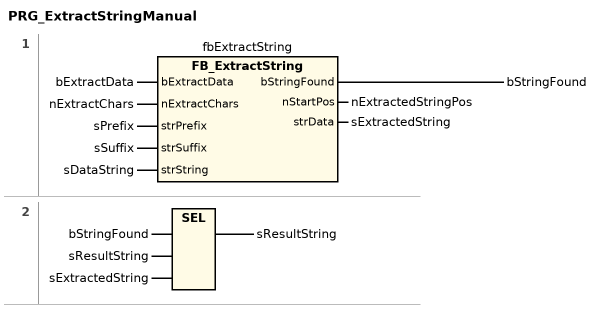
// NETWORK 1
fbExtractString(
    bExtractData := bExtractData,
    nExtractChars := nExtractChars,
    strPrefix := sPrefix,
    strSuffix := sSuffix,
    strString := sDataString,
    nStartPos => nExtractedStringPos,
    strData => sExtractedString); // FB_ExtractString
bStringFound := fbExtractString.bStringFound;

// NETWORK 2
sResultString := SEL(bStringFound, sResultString, sExtractedString);

END_PROGRAM

// ---- POUs/TcUnit/FUN_ReplaceLongSingleCharTests/PRG_ReplaceLongSingleCharManual.TcPOU
PROGRAM PRG_ReplaceLongSingleCharManual
VAR
	
	sFullCode		: T_LongSTRING := 'ST=53;$02CT=10;DS=GZDNP5JOA3IL$1D;OG=3;XP=-50;YP=50;AP=-88;CS=06.2;SC=0070;QS=3;PN=1;$03$04
											ST=53;$02CT=10;DS=N7E1Y89UNK3O$1D;OG=3;XP=-50;YP=-50;AP=-88;CS=06.2;SC=0070;QS=3;PN=2;$03$04
											ST=53;$02CT=10;DS=JHWJXYFNX9DS$1D;OG=3;XP=50;YP=50;AP=-88;CS=06.2;SC=0070;QS=3;PN=3;$03$04
											ST=53;$02CT=10;DS=XGBEZLBV8A9I$1D;OG=3;XP=50;YP=-50;AP=-88;CS=06.2;SC=0070;QS=3;PN=4;$03$04'; 
	sCharRemove		: T_Char := '$1D';
	sReplacmentChar	: T_Char := '';
	
	sResult			: T_LongSTRING;
END_VAR

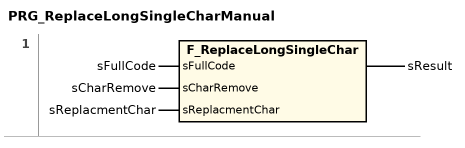
// NETWORK 1
sResult := F_ReplaceLongSingleChar(sFullCode := sFullCode, sCharRemove := sCharRemove, sReplacmentChar := sReplacmentChar);

END_PROGRAM

// ---- POUs/TcUnit/FB_LOGHandlerTests/PRG_LogHandlerManual.TcPOU
PROGRAM PRG_LogHandlerManual
VAR
	fbLogHandler			: FB_LOG_Handler;

	bLogData				: BOOL;
	sLogMessage				: T_LongSTRING;
	
	stEventDataUT				: ST_LOG_EventData;
	
	sResultMessage				: T_LongSTRING;
	
	bDone					: BOOL;
	bBufferOverflow			: BOOL;
END_VAR

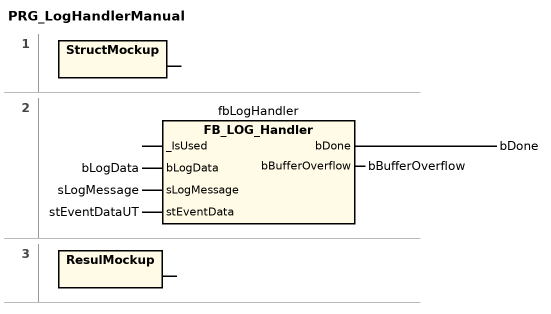
// NETWORK 1
StructMockup();

// NETWORK 2
fbLogHandler(
    bLogData := bLogData,
    sLogMessage := sLogMessage,
    stEventData := stEventDataUT,
    bBufferOverflow => bBufferOverflow); // FB_LOG_Handler
bDone := fbLogHandler.bDone;

// NETWORK 3
ResulMockup();

ACTION ResulMockup:
IF stEventDataUT.nImageByte < SIZEOF(sResultMessage) THEN
	MEMMOVE(ADR(sResultMessage), ADR(stEventDataUT.aDataLogImage), stEventDataUT.nImageByte);
END_IF
END_ACTION

ACTION StructMockup:

stEventDataUT.bEnable := gDevice.stMetsStatus.bSystemTimeValid;
stEventDataUT.sTimeStamp :=MID( F_SYSTEM_SystemTimeAsISO8601(gDevice.stMetsStatus.stCTDateTime.sSystemTime, gDevice.stMetsStatus.stCTDateTime.sUTCTimeZoneOffset ), 12, 12);

sLogMessage := '$01ST=53;$02CT=10;DS=GZDNP5JOA3IL;OG=3;XP=-50;YP=50;AP=-88;CS=06.2;SC=0070;QS=3;PN=1;$03
					$01ST=53;$02CT=10;DS=N7E1Y89UNK3O;OG=3;XP=-50;YP=-50;AP=-88;CS=06.2;SC=0070;QS=3;PN=2;$03
					$01ST=53;$02CT=10;DS=JHWJXYFNX9DS;OG=3;XP=50;YP=50;AP=-88;CS=06.2;SC=0070;QS=3;PN=3;$03
					$01ST=53;$02CT=10;DS=XGBEZLBV8A9I;OG=3;XP=50;YP=-50;AP=-88;CS=06.2;SC=0070;QS=3;PN=4;$03';
END_ACTION

END_PROGRAM

// ---- POUs/METS/Common LIB/08_SOFTWARE LIB/AI Codes And Validation FBs/F_CODE_GetItemAI.TcPOU
FUNCTION F_CODE_GetItemAI : T_MaxString
VAR_INPUT
	sFullCode		: T_MaxString;
	eCodeType		: E_CodeAI;
	stCodeInfo		: ST_CodeInfo;
END_VAR
VAR
	stItem			: ST_CodeValidation;
	
	sTemp			: T_MaxString;
	nStart			: INT;
	nEnd			: INT;
	
	sResultString	: T_MaxString;
END_VAR

IF stCodeInfo.nEntireLength > 0 THEN

	IF eCodeType = E_CodeAI.GTIN THEN 			stItem := stCodeInfo.stGTIN;
	ELSIF eCodeType = E_CodeAI.BATCH THEN 		stItem := stCodeInfo.stBatchID;
	ELSIF eCodeType = E_CodeAI.SERIAL THEN		stItem := stCodeInfo.stSerialCode;
	ELSIF eCodeType = E_CodeAI.PO THEN			stItem := stCodeInfo.stProductionOrder;
	ELSIF eCodeType = E_CodeAI.CRYPTO THEN		stItem := stCodeInfo.stCryptoCode;
	ELSIF eCodeType = E_CodeAI.RSKU THEN		stItem := stCodeInfo.stRSKU;
	ELSIF eCodeType = E_CodeAI.MRP THEN			stItem := stCodeInfo.stMRP;
	ELSIF eCodeType = E_CodeAI.BRANDSPEC THEN	stItem := stCodeInfo.stBrandSpecification;
	ELSIF eCodeType = E_CodeAI.PRODDATE THEN	stItem := stCodeInfo.stProduceDate;
	ELSIF eCodeType = E_CodeAI.USERFIELD THEN	stItem := stCodeInfo.stUserField3;
	END_IF

/////////////////////////////////////////////////////////////////////////////////////////////////////

	IF stItem.sStartAI <> '' AND stItem.sEndAI <> '' THEN
		
		nStart := FIND(sFullCode, stItem.sStartAI) + LEN(stItem.sStartAI);
		
		IF nStart > 0 THEN
			sTemp := RIGHT(sFullCode, LEN(sFullCode) - (nStart - 1));
		ELSE
			sTemp := sFullCode;
		END_IF
		
		nEnd := FIND(sTemp, stItem.sEndAI);
		
		IF nEnd = 0 THEN
			nEnd := LEN(sFullCode)+1;
		ELSE
			nEnd := nEnd +(nStart - 1);
		END_IF
		
	ELSIF stItem.sStartAI <> '' AND stItem.nCodeLength > 0 THEN
		
		nStart := FIND(sFullCode, stItem.sStartAI) + LEN(stItem.sStartAI);
		nEnd := nStart + stItem.nCodeLength;
		
	ELSIF stItem.nCodeStartPos > 0 AND stItem.sEndAI <> '' THEN
		
		nStart := stItem.nCodeStartPos;
		sTemp := RIGHT(sFullCode, LEN(sFullCode) - (nStart - 1));
		nEnd := FIND(sTemp, stItem.sEndAI);
		
		IF nEnd = 0 THEN
			nEnd := LEN(sFullCode)+1;
		ELSE
			nEnd := nEnd +(nStart - 1);
		END_IF
		
	ELSIF stItem.nCodeStartPos >= 0 AND stItem.nCodeLength > 0 THEN
		
		nStart := stItem.nCodeStartPos;
		nEnd := nStart + stItem.nCodeLength;
	ELSE
		nStart := 0;
		nEnd := 0;
	END_IF
	
	IF nStart > 0 AND nEnd > 0 THEN
		sResultString := MID(sFullCode, nEnd - nStart, nStart);
	ELSE
		sResultString := '';
	END_IF
ELSE
	sResultString := '';
END_IF

F_CODE_GetItemAI := sResultString;

END_FUNCTION

// ---- POUs/METS/Common LIB/09_SYSTEM LIB/FB_SYSTEM_CoreFolders.TcPOU
FUNCTION_BLOCK FB_SYSTEM_CoreFolders
VAR_INPUT
	bExecute				: BOOL;		(* set TRUE to generate system folders *)
	sBasePath			: T_FolderName;	(* CaseTrace base folder path *)
	aBaseFolder			: ARRAY[1..cSYSTEM_FOLDER_LIMIT] OF T_FolderName;
END_VAR
VAR_OUTPUT
	bDone				: BOOL;		(* TRUE = system folders complete *)
	bBusy				: BOOL;		(* TRUE = system folders in progress *)
	bError				: BOOL;		(* TRUE = system folders error *)
	nErrorID				: UDINT;	(* error code *)
	bSystemFolderOK		: BOOL;		(* TRUE = system folders OK *)
	sStatus					: STRING(25);	(* system folder status *)

END_VAR
VAR
	fbExecute				: R_TRIG;
	eState				: E_SYSTEM_MaintainFolders;
	eErrorState			: E_SYSTEM_MaintainFolders;
	nMaxIndex			: INT;
	nIndex				: INT;
	eCmdType		: E_EnumCmdType;
	fbFindFolder		: FB_EnumFindFileEntry;
	fbCreateFolder			: FB_CreateDir;

END_VAR

(* rising edge of bExecute *)
fbExecute(CLK := bExecute);

CASE eState OF

	(* idle *)
	E_FOLDER_IDLE:

		(* rising edge of bExecute *)
		IF fbExecute.Q = TRUE THEN

			(* update outputs *)
			bDone := FALSE;
			bBusy := TRUE;
			bError := FALSE;
			nErrorID := 0;

			(* max number of BASE folders and start with 1st folder *)
			nMaxIndex := UDINT_TO_INT(SIZEOF(aBaseFolder) / SIZEOF(aBaseFolder[1]));
			nIndex := 1;
			eCmdType := eEnumCmd_First;

			//eState := E_FOLDER_CREATEBASEPATH;
			eState := E_FOLDER_ININT_CHECK;

		(* bExecute has been reset *)
		ELSIF bExecute = FALSE THEN

			(* reset outputs *)
			bDone := FALSE;
			bBusy := FALSE;
			bError := FALSE;
			nErrorID := 0;
		END_IF

	E_FOLDER_ININT_CHECK:
					eCmdType := eEnumCmd_First;
					eState := E_FOLDER_CHECK;
	
	E_FOLDER_CHECK:

		(* find folder *)
		fbFindFolder(
			sNetId		:= '',
			sPathName	:= CONCAT(sBasePath, aBaseFolder[nIndex]),
			eCmd		:= eCmdType,
			bExecute	:= TRUE,
			tTimeout	:= T#1s
		);

		(* find folder complete *)
		IF fbFindFolder.bBusy = FALSE THEN

			(* find folder completed OK *)
			IF fbFindFolder.bError = FALSE THEN

				(* folder found *)
				IF fbFindFolder.stFindFile.fileAttributes.bDirectory = TRUE THEN

				
						(* all BASE folders completed *)
				IF nIndex = nMaxIndex THEN

					eState := E_FOLDER_DONE;

				(* more BASE folders *)
				ELSE
					nIndex := nIndex + 1;
					eCmdType := eEnumCmd_Abort;
					eState := E_FOLDER_ININT_CHECK;
				END_IF

				(* end of list *)
				ELSIF fbFindFolder.bEOE = TRUE THEN

						eState := E_FOLDER_CREATEBASEPATH;
				END_IF

			(* find folder completed OK *)
			ELSE

				(* update outputs *)
				bError := TRUE;
				nErrorID := fbFindFolder.nErrID;
				eErrorState := eState;

				eState := E_FOLDER_DONE;
			END_IF

			(* close off fbFindFolder *)
			fbFindFolder(bExecute := FALSE);
		END_IF
		
	(* create BASE folders *)
	E_FOLDER_CREATEBASEPATH:

		(* create folder *)
		fbCreateFolder(
			sNetId		:= '',
			sPathName	:= CONCAT(sBasePath, aBaseFolder[nIndex]),
			ePath		:= PATH_GENERIC,
			bExecute	:= TRUE,
			tTimeout	:= T#1s
		);

		(* create folder complete *)
		IF fbCreateFolder.bBusy = FALSE THEN

			(* create folder completed OK or folder already exists *)
			IF fbCreateFolder.bError = FALSE OR (fbCreateFolder.bError = TRUE AND fbCreateFolder.nErrId = cFAILED_OBJECT_ALREADY_EXIST) THEN

				(* all BASE folders completed *)
				IF nIndex = nMaxIndex THEN

					eState := E_FOLDER_DONE;

				(* more BASE folders *)
				ELSE

					(* next BASE folder *)
					nIndex := nIndex + 1;
					eState := E_FOLDER_ININT_CHECK;
				END_IF

			(* create folder error *)
			ELSE

				(* no error active *)
				IF bError = FALSE THEN

					(* update outputs *)
					bError := TRUE;
					nErrorID := fbCreateFolder.nErrId;
					eErrorState := eState;
					sStatus := CONCAT(sBasePath, aBaseFolder[nIndex]);
				END_IF

				eState := E_FOLDER_DONE;
			END_IF

			(* close off fbCreateFolder *)
			fbCreateFolder(bExecute := FALSE);
		END_IF


	(* done *)
	E_FOLDER_DONE:

		(* no error occurred *)
		IF bError = FALSE THEN

			(* update status *)
			bSystemFolderOK 		:= TRUE;
			sStatus 				:= 'Core folders OK';
			
		ELSE
			(* update status *)
			bSystemFolderOK 		:= FALSE;
			sStatus 				:= 'Core folders NOT OK';
		END_IF

		(* update outputs *)
		bDone := TRUE;
		bBusy := FALSE;

		eState := E_FOLDER_IDLE;


(* unknown state *)
ELSE

	eState := E_FOLDER_IDLE;

	(* reset outputs *)
	bDone := FALSE;
	bBusy := FALSE;
	bError := FALSE;
	nErrorID := 0;
	bSystemFolderOK := FALSE;
	sStatus := '';
END_CASE

END_FUNCTION_BLOCK

// ---- POUs/METS/Common LIB/09_SYSTEM LIB/FB_SYSTEM_CorePaths.TcPOU
FUNCTION_BLOCK FB_SYSTEM_CorePaths
VAR_INPUT
	bExecute				: BOOL;		(* set TRUE to generate system folders *)
	sMETSAppPath				: T_FolderPath;
	sMETSLogsPath				: T_FolderPath;	
	sMETSProcessPath			: T_FolderPath;
	aCoreFolders			: ARRAY[1..cSYSTEM_FOLDER_LIMIT] OF T_FolderName;
	aAuxFolders				: ARRAY[1..cSYSTEM_FOLDER_LIMIT] OF T_FolderName;
END_VAR
VAR_OUTPUT
	sArchiveDBPath			: T_FolderPath;	(*local ArchiveDB path*)
	sBridgeAppPath 			: T_FolderPath;	(* local Bridge path *)
	sLoggerAppPath			: T_FolderPath;	(*  *)
	sWebHMIPath				: T_FolderPath;	(*  *)
	sDeleteArchivePath		: T_FolderPath;	(*  *)
	
	sPCMPath 			: T_FolderPath;	(* local PCM path *)
	sPCMIncomingPath 	: T_FolderPath;	(* local PCM/Incoming path *)
	sCHMPath 			: T_FolderPath;	(* local CHM path *)
	sSettingsPath		 	: T_FolderPath;	(* local Setting*)
	sBackupsPath			: T_FolderPath; (*local Setting/Backup path*)
	sRecipePath				: T_FolderPath; (*local Setting/Recipe path*)
	sCamerasPath				: T_FolderPath;	(* local Camera path *)
	sPrintersPath			: T_FolderPath;	(* local Camera path *)
	
	sOCVPath 			: T_FolderPath;	(* local OCV path *)
	sOACPath 			: T_FolderPath;	(* local OAC path *)
	sCACPath 			: T_FolderPath;	(* local CAC path *)
	sSystemLogPath			: T_FolderPath;	(* local Log path *)
	
END_VAR
VAR
	fbExecute				: R_TRIG;

END_VAR
(*
cMETS_CORE_FOLDERS					: ARRAY[1..cSYSTEM_FOLDER_LIMIT] OF T_FolderName :=[
			(*01*)'CHM\',		(*02*)'CHM\Archive\',		(*03*)'CHM\Error\',		(*04*)'CHM\OK\',		(*05*)'CHM\Commissioning_Mode\',	(*06*)'CHM\Restore\',
			(*07*)'PCM\',		(*08*)'PCM\Archive\',		(*09*)'PCM\Error\',		(*10*)'PCM\Incoming\',
			(*11*)'Settings\',	(*12*)'Settings\Backups\',	(*13*)'Settings\Recipe\',
			(*14*)'Cameras\',
			(*15*)'Printers\',	(*16*)'Printers\Templates'];
			
cMETS_AUX_FOLDERS					: ARRAY[1..cSYSTEM_FOLDER_LIMIT] OF T_FolderName :=[
			(*01*)'CAC\',		(*02*)'CAC\Archive\',		(*03*)'CAC\Error\',		(*04*)'CAC\Restored\',
			(*05*)'OAC\',		(*06*)'OAC\Error\',			(*07*)'OAC\Empty\',
			(*08*)'OCV\',		(*09*)'OCV\Error\',			(*10*)'OCV\Empty\',
			(*11*)'SystemLog\',
			(*12*)'ArchiveDB\',
			(*13*)'BridgeApp\Bridge_Core\',
			(*14*)'LoggerApp\Service\',
			(*15*)'WebHMI\',
			(*16*)'DeleteArchiveTool\'];
*)


(* rising edge of bExecute *)
fbExecute(CLK := bExecute);

(* rising edge of bExecute *)
IF fbExecute.Q = TRUE THEN

(* populate local folder paths *)
	sArchiveDBPath			:= CONCAT(sMETSAppPath, aAuxFolders[12]);
	sBridgeAppPath 			:= CONCAT(sMETSAppPath, aAuxFolders[13]);
	sLoggerAppPath			:= CONCAT(sMETSAppPath, aAuxFolders[14]);
	sWebHMIPath				:= CONCAT(sMETSAppPath, aAuxFolders[15]);
	sDeleteArchivePath		:= CONCAT(sMETSAppPath, aAuxFolders[16]);
	
	sPCMPath 				:= CONCAT(sMETSProcessPath, aCoreFolders[7]);
	sPCMIncomingPath 		:= CONCAT(sMETSProcessPath, aCoreFolders[10]);
	sCHMPath 				:= CONCAT(sMETSProcessPath, aCoreFolders[1]);
	sSettingsPath		 	:= CONCAT(sMETSProcessPath, aCoreFolders[11]);
	sBackupsPath			:= CONCAT(sMETSProcessPath, aCoreFolders[12]);
	sRecipePath				:= CONCAT(sMETSProcessPath, aCoreFolders[13]);
	sCamerasPath			:= CONCAT(sMETSProcessPath, aCoreFolders[14]);
	sPrintersPath			:= CONCAT(sMETSProcessPath, aCoreFolders[15]);
	
	sOCVPath 				:= CONCAT(sMETSProcessPath, aAuxFolders[8]);
	sOACPath 				:= CONCAT(sMETSProcessPath, aAuxFolders[5]);
	sCACPath 				:= CONCAT(sMETSProcessPath, aAuxFolders[1]);
	
	sSystemLogPath			:= CONCAT(sMETSLogsPath, aAuxFolders[11]);
			
ELSIF NOT bExecute THEN		
			
	(* populate local folder paths *)
	sArchiveDBPath			:='';
	sBridgeAppPath 			:='';
	sLoggerAppPath			:='';
	sWebHMIPath				:='';
	sDeleteArchivePath		:='';
	
	sPCMPath 				:='';
	sPCMIncomingPath 		:='';
	sCHMPath 				:='';
	sSettingsPath		 	:='';
	sBackupsPath			:='';
	sRecipePath				:='';
	sCamerasPath			:='';
	sPrintersPath			:='';
	
	sOCVPath 				:='';
	sOACPath 				:='';
	sCACPath 				:='';
	
	sSystemLogPath			:='';		
			
END_IF

END_FUNCTION_BLOCK

// ---- POUs/TcUnit/FB_CASE_ValidateContentTests/PRG_CASE_ValidateContentManual.TcPOU
PROGRAM PRG_CASE_ValidateContentManual
VAR
	fbCase_ValidateContent		: FB_CASE_ValidateContent;
	
	
	(* Init function/method declarations*)
	rTrigDataInit		: R_TRIG;
	bDataInit			: BOOL;
	iOuter				: INT;
	iPack				: INT;
	sPackNum			: STRING;
	sOuterNum			: STRING;
	sPackCode			: STRING;
	
	(* Inputs *)
	bExecute 					: BOOL;
	stCTDateTime				: ST_SYSTEM_DateTime;	(* CaseTrace date/time structure *)
	bIsDuplicateOuters			: BOOL;
	bIsDuplicatePacks			: BOOL;
	stOuterDataNotFound			: ST_RejectItems;
	stRejectReasonsForOuter		: ST_RejectReasonsForOuter;
	
	(* In/Out *)
	stProductInstruction		: ST_PCM_Status;
	nSecquentionalCounter		: UDINT;
	stCodeInfo_Outer			: ST_CodeInfo;
	stCaseRejectReasons			: ST_RejectReasonsForCase;
	stCACData 					: ST_CAC_Data;
	
	(* Outputs *)
	bDone 						: BOOL;
	bBusy						: BOOL;
	bError						: BOOL;
	nErrorID 					: UDINT;

	sRejectCode					: T_MaxString;
	nValidationIndex			: INT;
	
END_VAR

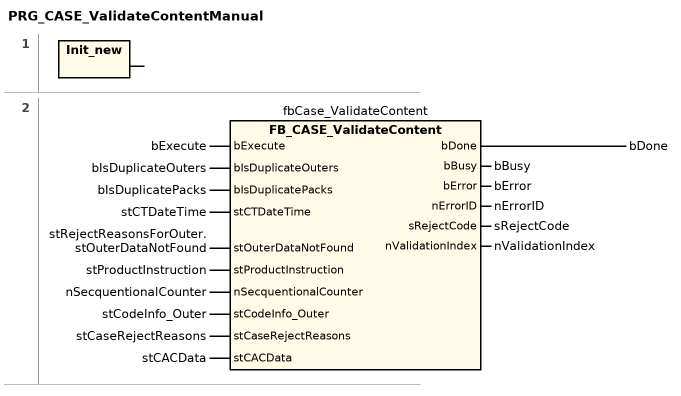
// NETWORK 1
Init_new();

// NETWORK 2
fbCase_ValidateContent(
    bExecute := bExecute,
    bIsDuplicateOuters := bIsDuplicateOuters,
    bIsDuplicatePacks := bIsDuplicatePacks,
    stCTDateTime := stCTDateTime,
    stOuterDataNotFound := stRejectReasonsForOuter.stOuterDataNotFound,
    stProductInstruction := stProductInstruction,
    nSecquentionalCounter := nSecquentionalCounter,
    stCodeInfo_Outer := stCodeInfo_Outer,
    stCaseRejectReasons := stCaseRejectReasons,
    stCACData := stCACData,
    bBusy => bBusy,
    bError => bError,
    nErrorID => nErrorID,
    sRejectCode => sRejectCode,
    nValidationIndex => nValidationIndex); // FB_CASE_ValidateContent
bDone := fbCase_ValidateContent.bDone;

ACTION Init:
rTrigDataInit(CLK := bDataInit);

IF rTrigDataInit.Q THEN
		
	stProductInstruction.nOutersPerCase		:= 50;
	stProductInstruction.nPacksPerOuter 	:= 10;











	FOR iOuter := 1 TO stProductInstruction.nOutersPerCase DO
		(* Ustaw outer *)
		stCACData.Outer[iOuter].Barcode    := CONCAT('OUTER', INT_TO_STRING(iOuter));
		stCACData.Outer[iOuter].OuterCodeStatus := 5;
		






		FOR iPack := 1 TO stProductInstruction.nPacksPerOuter DO
			(* Pack number z zerami *)
			sPackNum := CONCAT('0', INT_TO_STRING(iPack));  (* dla 1-9: '01'-'09' *)
			IF iPack = 10 THEN
				sPackNum := '10';
			END_IF;
			
			(* Outer number z zerami dla 1-9 *)
			sOuterNum := CONCAT('0', INT_TO_STRING(iOuter));
			IF iOuter >= 10 THEN
				sOuterNum := INT_TO_STRING(iOuter);
			END_IF;
			
			(* Sklej pack code *)
			sPackCode := CONCAT(CONCAT('PACK', sPackNum), CONCAT('OUTER', sOuterNum));
			
			(* Przypisz *)
			stCACData.Outer[iOuter].PackCode[iPack]			:= sPackCode;
			stCACData.Outer[iOuter].PackCodeStatus[iPack]	:= 5;
			stCACData.Outer[iOuter].PackRejectID[iPack]		:= 0;


			
		END_FOR;
	END_FOR;	










	
END_IF
END_ACTION

ACTION Init_new:

rTrigDataInit(CLK := bDataInit);

IF rTrigDataInit.Q THEN
	
	MEMSET(ADR(stCACData), 16#00, SIZEOF(stCACData));	
	
	stProductInstruction.nOutersPerCase 	:= 50;
	stProductInstruction.nPacksPerOuter		:= 10;	
	// jezeli tej wartosci nie ma, jest na 0 i czytaj ponizej
	stProductInstruction.nPacksPerCase		:= 500;
	stProductInstruction.nOpMode			:= 11;
	stProductInstruction.sRetailSKU			:= '1234567';
	stProductInstruction.nAcceptanceLevel 	:= 10;

	// jezeli stCACData.NumberOfOuters=0 , czyli usune te linie ponizej to nie wejdzie do warunku linia 40 FB_CASE_ValidateContent i wywali
	// jakis error z elsifa ktoregos
	stCACData.NumberOfOuters			:= stProductInstruction.nOutersPerCase;
	stCACData.CodingAndTrackingMode		:= stProductInstruction.nOpMode;
	stCACData.RetailSKU					:= stProductInstruction.sRetailSKU;

	FOR iOuter := 1 TO stProductInstruction.nOutersPerCase DO
		(* Outer number z zerami *)
		sOuterNum := F_StringAddPrefix(INT_TO_STRING(iOuter),2,'0');
	
		stCACData.Outer[iOuter].Barcode    				:= CONCAT('OUTER', sOuterNum);
		stCACData.Outer[iOuter].NumberOfPacks 			:= stProductInstruction.nPacksPerOuter;
		stCACData.Outer[iOuter].NumberOfLinkedPacks 	:= stProductInstruction.nPacksPerOuter;
		stCACData.Outer[iOuter].AcceptanceLevel 		:= stProductInstruction.nAcceptanceLevel;
		stCACData.Outer[iOuter].CodingAndTrackingMode	:= stProductInstruction.nOpMode;
		stCACData.Outer[iOuter].OuterRejectCode			:= 'OK';
	
		FOR iPack := 1 TO stProductInstruction.nPacksPerOuter DO
			(* Pack number dwucyfrowy z zerami *)
			sPackNum := F_StringAddPrefix(INT_TO_STRING(iPack),2,'0');			
			(* Sklej pack code *)
			sPackCode := CONCAT(CONCAT('PACK', sPackNum), CONCAT('OUTER', sOuterNum));
			
			(* Write Pack Barcodes / Data*)
			stCACData.Outer[iOuter].PackCode[iPack]				:= sPackCode;
			stCACData.Outer[iOuter].PackCodeStatus[iPack]		:= 5;
			stCACData.Outer[iOuter].PackRejectID[iPack]			:= 0;			
			stCACData.Outer[iOuter].PackRejectCode[iPack]		:= 'OK';			
			stCACData.Outer[iOuter].PackCodeStatus[iPack].5 	:= TRUE;
			
			
			IF iPack = 1 THEN
				stCACData.Outer[iOuter].AggregationCodes[1]	:= stCACData.Outer[iOuter].PackCode[iPack];
			END_IF
			IF iPack = 2 THEN
				stCACData.Outer[iOuter].AggregationCodes[2]	:= stCACData.Outer[iOuter].PackCode[iPack];
			END_IF
		END_FOR
	END_FOR	
	
	stCACData.Outer[3].OuterCodeStatus.5 	:= TRUE;
	stCACData.Outer[4].OuterCodeStatus.5	:= TRUE;
	
	stCACData.NumberOfOuters 				:= 55;
	
END_IF
END_ACTION

END_PROGRAM

// ---- POUs/_Exclude/F13_CaseContentValidation_ORG.TcPOU
PROGRAM F13_CaseContentValidation_ORG
VAR
	fbCrossPushCounter					: CTU;
	bCaseCompleteInsidePacker			: BOOL;


	rtrigSetEarlyCaseValidationOK			: R_TRIG;
	rtrigSetEarlyCaseValidationNOK		: R_TRIG;

	fbBiuldPackerLogString				: FB_CASE_BiuldPackerLogString;
	fbShiftPackerQueue					: FB_CASE_ShiftPackerQueue;
	fbMovePackerToCase				: FB_CASE_MovePackerToCase;
	fbFinaliseCaseData					: FB_CASE_FinaliseCaseData;

	fbValidationIndexOK					: FB_CTU32;
	fbValidationIndexNoData				: FB_CTU32;
	fbValidationIndexUnder				: FB_CTU32;
	fbValidationIndexOver				: FB_CTU32;


	fbDebugCNT				: FB_DEBUG_CounterArray;
	aCNTDebug				: ARRAY [1..10] OF UDINT;
	bResetCNT					: BOOL;


END_VAR

(*
Modification history:
Date		|	Author 		|	Remark
----------------------------------------------------------------------------------------------------
02.09.20	|	PP			|	Start Remarking.
*)

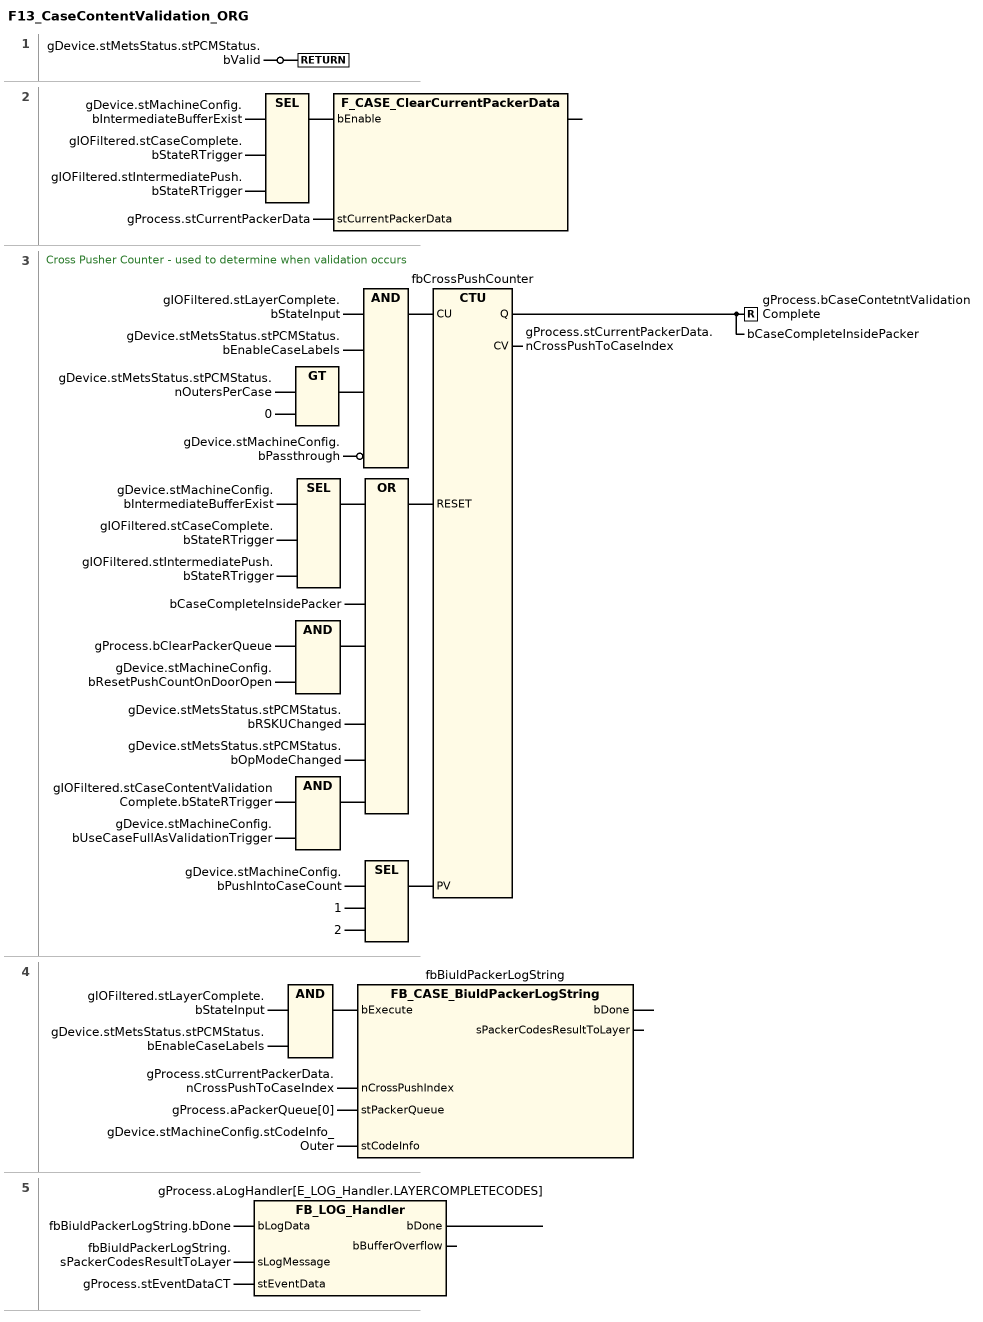
// NETWORK 1
IF NOT gDevice.stMetsStatus.stPCMStatus.bValid THEN RETURN; END_IF

// NETWORK 2
F_CASE_ClearCurrentPackerData(bEnable := SEL(gDevice.stMachineConfig.bIntermediateBufferExist, gIOFiltered.stCaseComplete.bStateRTrigger, gIOFiltered.stIntermediatePush.bStateRTrigger), stCurrentPackerData := gProcess.stCurrentPackerData);

// NETWORK 3
// 					Cross Pusher Counter - used to determine when validation occurs
//
//
fbCrossPushCounter(
    CU := gIOFiltered.stLayerComplete.bStateInput AND gDevice.stMetsStatus.stPCMStatus.bEnableCaseLabels AND gDevice.stMetsStatus.stPCMStatus.nOutersPerCase > 0 AND NOT gDevice.stMachineConfig.bPassthrough,
    RESET := SEL(gDevice.stMachineConfig.bIntermediateBufferExist, gIOFiltered.stCaseComplete.bStateRTrigger, gIOFiltered.stIntermediatePush.bStateRTrigger) OR bCaseCompleteInsidePacker OR gProcess.bClearPackerQueue AND gDevice.stMachineConfig.bResetPushCountOnDoorOpen OR gDevice.stMetsStatus.stPCMStatus.bRSKUChanged OR gDevice.stMetsStatus.stPCMStatus.bOpModeChanged OR gIOFiltered.stCaseContentValidationComplete.bStateRTrigger AND gDevice.stMachineConfig.bUseCaseFullAsValidationTrigger,
    PV := SEL(gDevice.stMachineConfig.bPushIntoCaseCount, 1, 2),
    CV => gProcess.stCurrentPackerData.nCrossPushToCaseIndex); // CTU
gProcess.bCaseContetntValidationComplete R= fbCrossPushCounter.Q;
bCaseCompleteInsidePacker := fbCrossPushCounter.Q;

// NETWORK 4
fbBiuldPackerLogString(
    bExecute := gIOFiltered.stLayerComplete.bStateInput AND gDevice.stMetsStatus.stPCMStatus.bEnableCaseLabels,
    nCrossPushIndex := gProcess.stCurrentPackerData.nCrossPushToCaseIndex,
    stPackerQueue := gProcess.aPackerQueue[0],
    stCodeInfo := gDevice.stMachineConfig.stCodeInfo_Outer); // FB_CASE_BiuldPackerLogString

// NETWORK 5
gProcess.aLogHandler[E_LOG_Handler.LAYERCOMPLETECODES](
    bLogData := fbBiuldPackerLogString.bDone,
    sLogMessage := fbBiuldPackerLogString.sPackerCodesResultToLayer,
    stEventData := gProcess.stEventDataCT); // FB_LOG_Handler

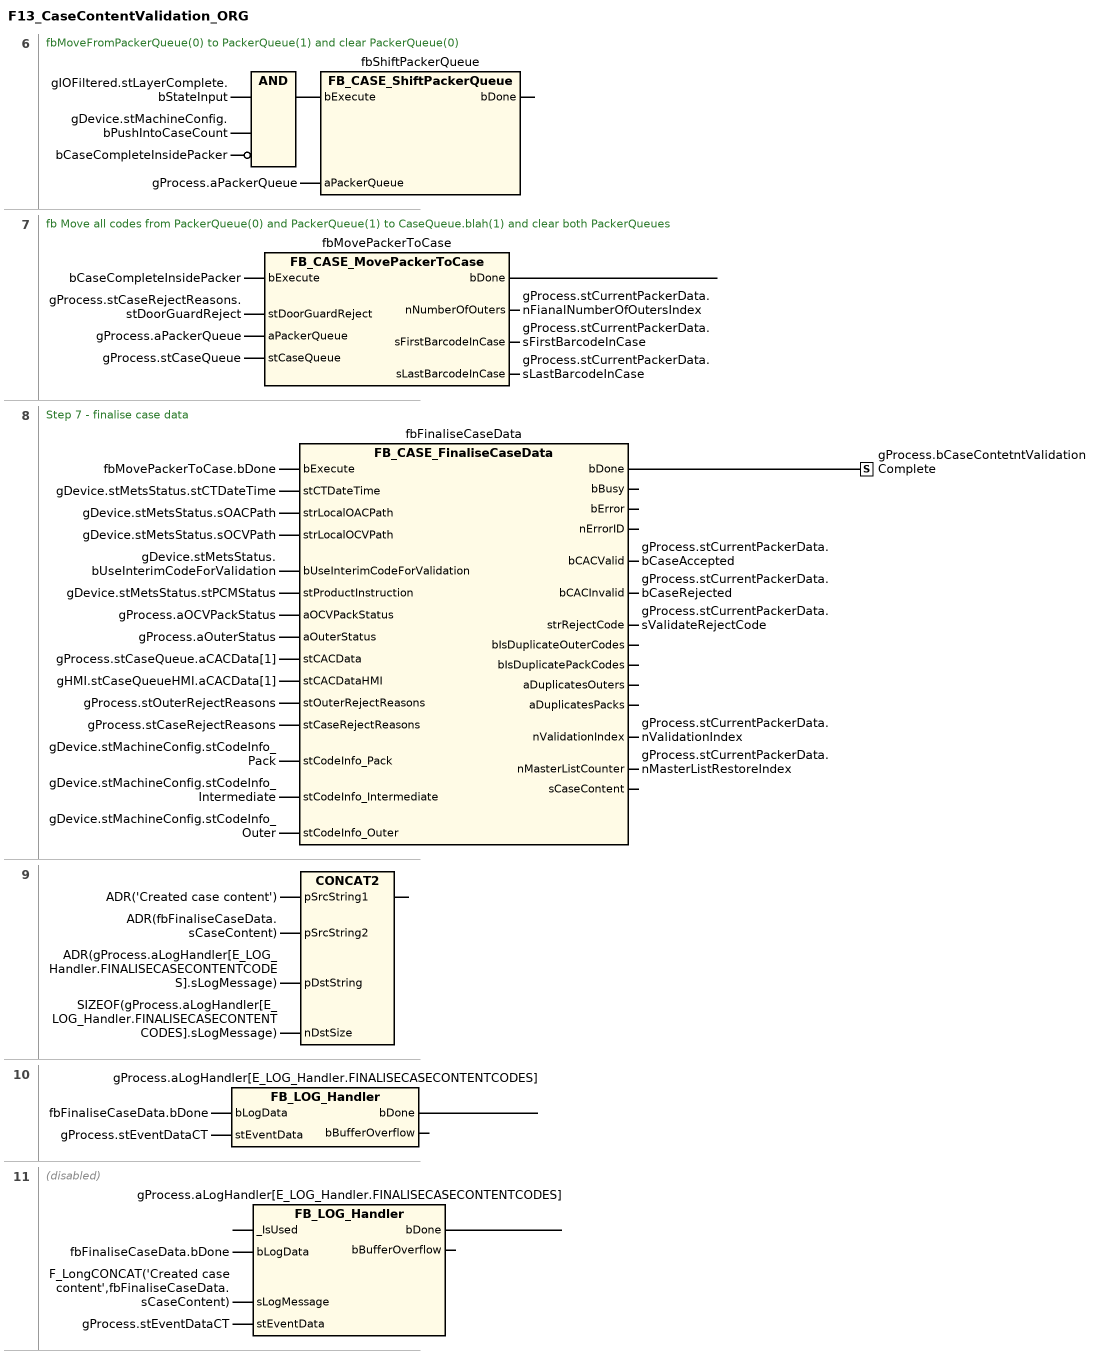
// NETWORK 6
// fbMoveFromPackerQueue(0) to PackerQueue(1) and clear PackerQueue(0)
fbShiftPackerQueue(bExecute := gIOFiltered.stLayerComplete.bStateInput AND gDevice.stMachineConfig.bPushIntoCaseCount AND NOT bCaseCompleteInsidePacker, aPackerQueue := gProcess.aPackerQueue); // FB_CASE_ShiftPackerQueue

// NETWORK 7
// fb Move all codes from PackerQueue(0) and PackerQueue(1) to CaseQueue.blah(1) and clear both PackerQueues
fbMovePackerToCase(
    bExecute := bCaseCompleteInsidePacker,
    stDoorGuardReject := gProcess.stCaseRejectReasons.stDoorGuardReject,
    aPackerQueue := gProcess.aPackerQueue,
    stCaseQueue := gProcess.stCaseQueue,
    nNumberOfOuters => gProcess.stCurrentPackerData.nFianalNumberOfOutersIndex,
    sFirstBarcodeInCase => gProcess.stCurrentPackerData.sFirstBarcodeInCase,
    sLastBarcodeInCase => gProcess.stCurrentPackerData.sLastBarcodeInCase); // FB_CASE_MovePackerToCase

// NETWORK 8
// Step 7 - finalise case data
fbFinaliseCaseData(
    bExecute := fbMovePackerToCase.bDone,
    stCTDateTime := gDevice.stMetsStatus.stCTDateTime,
    strLocalOACPath := gDevice.stMetsStatus.sOACPath,
    strLocalOCVPath := gDevice.stMetsStatus.sOCVPath,
    bUseInterimCodeForValidation := gDevice.stMetsStatus.bUseInterimCodeForValidation,
    stProductInstruction := gDevice.stMetsStatus.stPCMStatus,
    aOCVPackStatus := gProcess.aOCVPackStatus,
    aOuterStatus := gProcess.aOuterStatus,
    stCACData := gProcess.stCaseQueue.aCACData[1],
    stCACDataHMI := gHMI.stCaseQueueHMI.aCACData[1],
    stOuterRejectReasons := gProcess.stOuterRejectReasons,
    stCaseRejectReasons := gProcess.stCaseRejectReasons,
    stCodeInfo_Pack := gDevice.stMachineConfig.stCodeInfo_Pack,
    stCodeInfo_Intermediate := gDevice.stMachineConfig.stCodeInfo_Intermediate,
    stCodeInfo_Outer := gDevice.stMachineConfig.stCodeInfo_Outer,
    bCACValid => gProcess.stCurrentPackerData.bCaseAccepted,
    bCACInvalid => gProcess.stCurrentPackerData.bCaseRejected,
    strRejectCode => gProcess.stCurrentPackerData.sValidateRejectCode,
    nValidationIndex => gProcess.stCurrentPackerData.nValidationIndex,
    nMasterListCounter => gProcess.stCurrentPackerData.nMasterListRestoreIndex); // FB_CASE_FinaliseCaseData
gProcess.bCaseContetntValidationComplete S= fbFinaliseCaseData.bDone;

// NETWORK 9
CONCAT2(pSrcString1 := ADR('Created case content'), pSrcString2 := ADR(fbFinaliseCaseData.sCaseContent), pDstString := ADR(gProcess.aLogHandler[E_LOG_Handler.FINALISECASECONTENTCODES].sLogMessage), nDstSize := SIZEOF(gProcess.aLogHandler[E_LOG_Handler.FINALISECASECONTENTCODES].sLogMessage));

// NETWORK 10
gProcess.aLogHandler[E_LOG_Handler.FINALISECASECONTENTCODES](bLogData := fbFinaliseCaseData.bDone, stEventData := gProcess.stEventDataCT); // FB_LOG_Handler

// NETWORK 11 (disabled)
// gProcess.aLogHandler[E_LOG_Handler.FINALISECASECONTENTCODES](
//     bLogData := fbFinaliseCaseData.bDone,
//     sLogMessage := F_LongCONCAT('Created case content',fbFinaliseCaseData.sCaseContent),
//     stEventData := gProcess.stEventDataCT); // FB_LOG_Handler

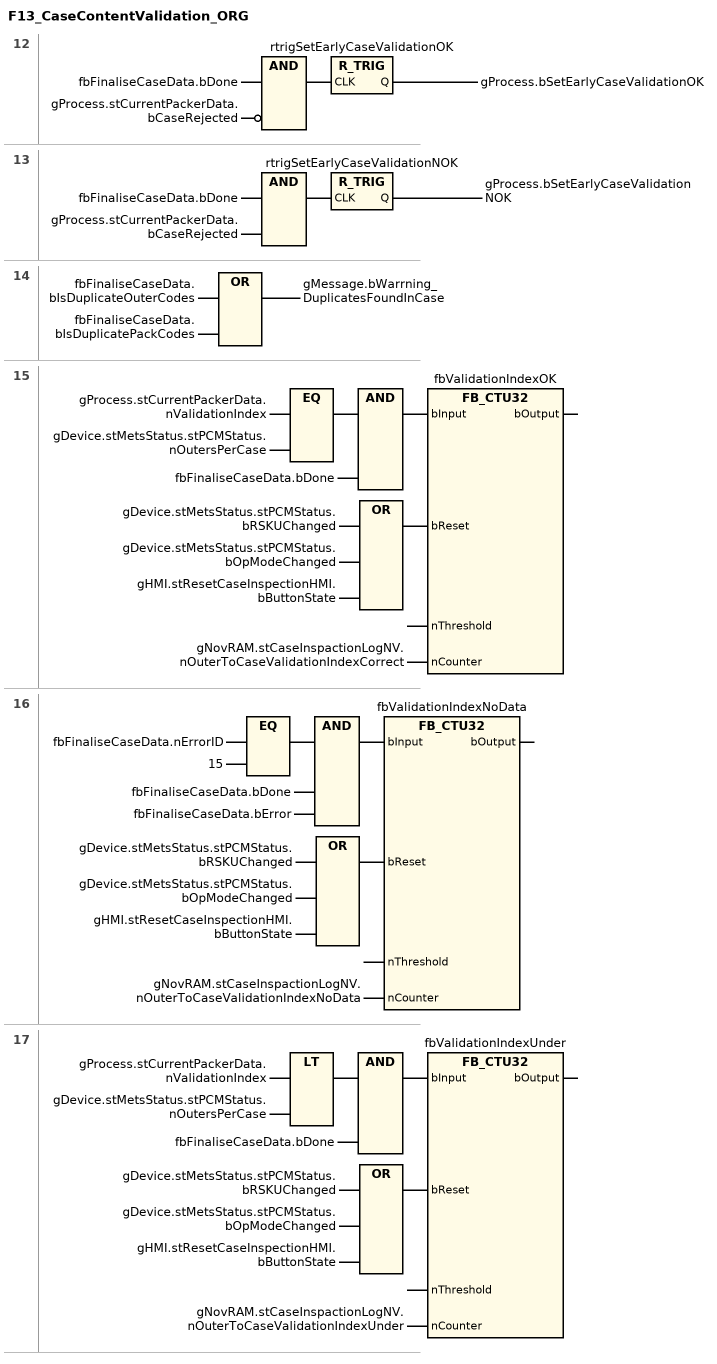
// NETWORK 12
rtrigSetEarlyCaseValidationOK(CLK := fbFinaliseCaseData.bDone AND NOT gProcess.stCurrentPackerData.bCaseRejected); // R_TRIG
gProcess.bSetEarlyCaseValidationOK := rtrigSetEarlyCaseValidationOK.Q;

// NETWORK 13
rtrigSetEarlyCaseValidationNOK(CLK := fbFinaliseCaseData.bDone AND gProcess.stCurrentPackerData.bCaseRejected); // R_TRIG
gProcess.bSetEarlyCaseValidationNOK := rtrigSetEarlyCaseValidationNOK.Q;

// NETWORK 14
gMessage.bWarrning_DuplicatesFoundInCase := fbFinaliseCaseData.bIsDuplicateOuterCodes OR fbFinaliseCaseData.bIsDuplicatePackCodes;

// NETWORK 15
fbValidationIndexOK(
    bInput := gProcess.stCurrentPackerData.nValidationIndex = gDevice.stMetsStatus.stPCMStatus.nOutersPerCase AND fbFinaliseCaseData.bDone,
    bReset := gDevice.stMetsStatus.stPCMStatus.bRSKUChanged OR gDevice.stMetsStatus.stPCMStatus.bOpModeChanged OR gHMI.stResetCaseInspectionHMI.bButtonState,
    nCounter := gNovRAM.stCaseInspactionLogNV.nOuterToCaseValidationIndexCorrect); // FB_CTU32

// NETWORK 16
fbValidationIndexNoData(
    bInput := fbFinaliseCaseData.nErrorID = 15 AND fbFinaliseCaseData.bDone AND fbFinaliseCaseData.bError,
    bReset := gDevice.stMetsStatus.stPCMStatus.bRSKUChanged OR gDevice.stMetsStatus.stPCMStatus.bOpModeChanged OR gHMI.stResetCaseInspectionHMI.bButtonState,
    nCounter := gNovRAM.stCaseInspactionLogNV.nOuterToCaseValidationIndexNoData); // FB_CTU32

// NETWORK 17
fbValidationIndexUnder(
    bInput := gProcess.stCurrentPackerData.nValidationIndex < gDevice.stMetsStatus.stPCMStatus.nOutersPerCase AND fbFinaliseCaseData.bDone,
    bReset := gDevice.stMetsStatus.stPCMStatus.bRSKUChanged OR gDevice.stMetsStatus.stPCMStatus.bOpModeChanged OR gHMI.stResetCaseInspectionHMI.bButtonState,
    nCounter := gNovRAM.stCaseInspactionLogNV.nOuterToCaseValidationIndexUnder); // FB_CTU32

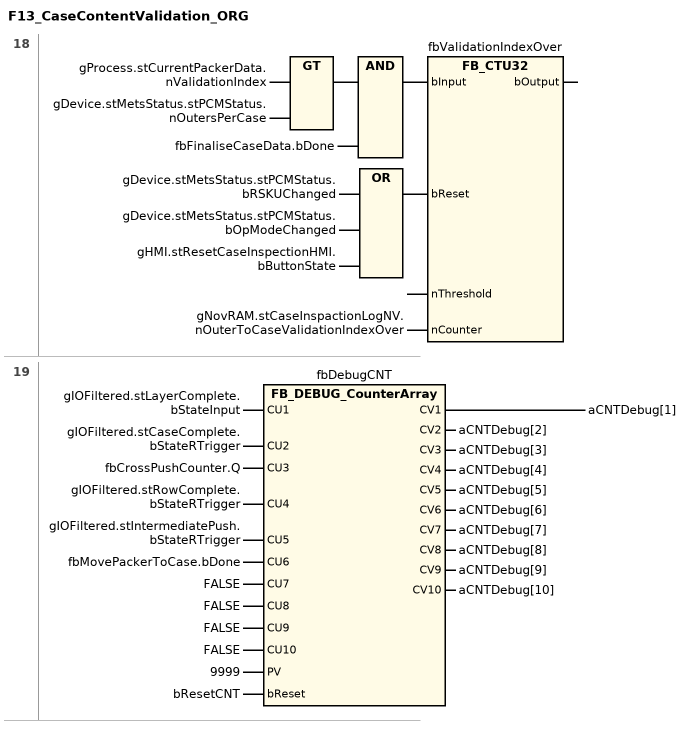
// NETWORK 18
fbValidationIndexOver(
    bInput := gProcess.stCurrentPackerData.nValidationIndex > gDevice.stMetsStatus.stPCMStatus.nOutersPerCase AND fbFinaliseCaseData.bDone,
    bReset := gDevice.stMetsStatus.stPCMStatus.bRSKUChanged OR gDevice.stMetsStatus.stPCMStatus.bOpModeChanged OR gHMI.stResetCaseInspectionHMI.bButtonState,
    nCounter := gNovRAM.stCaseInspactionLogNV.nOuterToCaseValidationIndexOver); // FB_CTU32

// NETWORK 19
fbDebugCNT(
    CU1 := gIOFiltered.stLayerComplete.bStateInput,
    CU2 := gIOFiltered.stCaseComplete.bStateRTrigger,
    CU3 := fbCrossPushCounter.Q,
    CU4 := gIOFiltered.stRowComplete.bStateRTrigger,
    CU5 := gIOFiltered.stIntermediatePush.bStateRTrigger,
    CU6 := fbMovePackerToCase.bDone,
    CU7 := FALSE,
    CU8 := FALSE,
    CU9 := FALSE,
    CU10 := FALSE,
    PV := 9999,
    bReset := bResetCNT,
    CV2 => aCNTDebug[2],
    CV3 => aCNTDebug[3],
    CV4 => aCNTDebug[4],
    CV5 => aCNTDebug[5],
    CV6 => aCNTDebug[6],
    CV7 => aCNTDebug[7],
    CV8 => aCNTDebug[8],
    CV9 => aCNTDebug[9],
    CV10 => aCNTDebug[10]); // FB_DEBUG_CounterArray
aCNTDebug[1] := fbDebugCNT.CV1;

END_PROGRAM

// ---- POUs/METS/Common LIB/04_CASE LIB/Case FBs/FB_CASE_BiuldPackerLogString.TcPOU
(* shifts specified group of cases from Packer layer 0 to Packer layer 1 *)
FUNCTION_BLOCK FB_CASE_BiuldPackerLogString
VAR_INPUT
	bExecute				: BOOL;			(* set TRUE to shift Case Queue *)
	nCrossPushIndex		: UINT;
END_VAR
VAR_IN_OUT
	stPackerQueue 			: ST_CASE_InfeedQueue;	(* Outfeed Queue *)
	stCodeInfo					: ST_CodeInfo;
END_VAR
VAR_OUTPUT
	bDone				: BOOL;			(* TRUE = complete *)
	sPackerCodesResultToLayer	: T_LongSTRING;
END_VAR
VAR
	fbExecute				: R_TRIG;
	nPackerLogIndex		: INT;
	sAppendedString		: STRING;
END_VAR

(* rising edge of bExecute *)
fbExecute(CLK:= bExecute);

(* move CaseData *)
IF fbExecute.Q = TRUE THEN
	
	sAppendedString				:= '';
	sPackerCodesResultToLayer 	:= '';

	sPackerCodesResultToLayer :=  F_CONCAT3('LayerComplete ', UINT_TO_STRING(nCrossPushIndex),' moved ');
	sPackerCodesResultToLayer := F_CONCAT4(sPackerCodesResultToLayer, '[', INT_TO_STRING(stPackerQueue.nIndex),']:');
	FOR nPackerLogIndex := 1 TO MIN(stPackerQueue.nIndex ,cMAX_INFEED_QUEUE) BY 1 DO
		
		//sPackerCodesResultToLayer :=F_LongCONCAT(sPackerCodesResultToLayer, '   ');
		//sPackerCodesResultToLayer := F_LongCONCAT(sPackerCodesResultToLayer, RIGHT(F_CODE_GetItem(stPackerQueue.aOuter[nPackerLogIndex].Barcode, eCodeAIType.SerialCode,  stCodeInfo),7));
		
		CONCAT2(ADR(sPackerCodesResultToLayer), ADR('   '), ADR(sPackerCodesResultToLayer), SIZEOF(sPackerCodesResultToLayer));
		
		sAppendedString := RIGHT(F_CODE_GetItem(stPackerQueue.aOuter[nPackerLogIndex].Barcode, eCodeAIType.SerialCode,  stCodeInfo),7);
		CONCAT2(ADR(sPackerCodesResultToLayer), ADR(sAppendedString), ADR(sPackerCodesResultToLayer), SIZEOF(sPackerCodesResultToLayer));

	END_FOR

	bDone := TRUE;

(* bExecute has been reset *)
ELSIF bExecute = FALSE THEN
	bDone := FALSE;
END_IF

END_FUNCTION_BLOCK

// ---- POUs/METS/Common LIB/08_SOFTWARE LIB/AI Codes And Validation FBs/F_CODE_GetItem.TcPOU
FUNCTION F_CODE_GetItem : T_MaxString
VAR_INPUT
	sFullCode			: T_MaxString;
	nCodeType		: INT;
	stCodeInfo		: ST_CodeInfo;
END_VAR
VAR
	stItem			: ST_CodeValidation;
	eCodeAIPattern	: E_CodeAIType;
	sItem			: T_MaxString;
	nStart			: INT;
	nEnd				: INT;
	sTemp			: T_MaxString;
END_VAR

IF stCodeInfo.nEntireLength > 0 THEN

	IF nCodeType = eCodeAIPattern.GTIN THEN 				stItem := stCodeInfo.stGTIN;
	ELSIF nCodeType = eCodeAIPattern.BatchID THEN 		stItem := stCodeInfo.stBatchID;
	ELSIF nCodeType = eCodeAIPattern.SerialCode THEN		stItem := stCodeInfo.stSerialCode;
	ELSIF nCodeType = eCodeAIPattern.ProductionOrder THEN	stItem := stCodeInfo.stProductionOrder;
	ELSIF nCodeType = eCodeAIPattern.CryptoCode THEN		stItem := stCodeInfo.stCryptoCode;
	ELSIF nCodeType = eCodeAIPattern.RSKU THEN			stItem := stCodeInfo.stRSKU;
	ELSIF nCodeType = eCodeAIPattern.MRP THEN			stItem := stCodeInfo.stMRP;
	ELSIF nCodeType = eCodeAIPattern.BrandSpecification THEN		stItem := stCodeInfo.stBrandSpecification;
	ELSIF nCodeType = eCodeAIPattern.ProduceDate THEN		stItem := stCodeInfo.stProduceDate;
	ELSIF nCodeType = eCodeAIPattern.UserField3 THEN		stItem := stCodeInfo.stUserField3;
	END_IF


	IF stItem.sStartAI <> '' AND stItem.sEndAI <> '' THEN
		nStart := FIND(sFullCode, stItem.sStartAI) + LEN(stItem.sStartAI);
		IF nStart > 0 THEN
			sTemp := RIGHT(sFullCode, LEN(sFullCode) - (nStart - 1));
		ELSE
			sTemp := sFullCode;
		END_IF
		nEnd := FIND(sTemp, stItem.sEndAI);
		IF nEnd = 0 THEN
			nEnd := LEN(sFullCode)+1;
		ELSE
			nEnd := nEnd +(nStart - 1);
		END_IF
	ELSIF stItem.sStartAI <> '' AND stItem.nCodeLength > 0 THEN
		nStart := FIND(sFullCode, stItem.sStartAI) + LEN(stItem.sStartAI);
		nEnd := nStart + stItem.nCodeLength;
	ELSIF stItem.nCodeStartPos > 0 AND stItem.sEndAI <> '' THEN
		nStart := stItem.nCodeStartPos;
		sTemp := RIGHT(sFullCode, LEN(sFullCode) - (nStart - 1));
		nEnd := FIND(sTemp, stItem.sEndAI);
		IF nEnd = 0 THEN
			nEnd := LEN(sFullCode)+1;
		ELSE
			nEnd := nEnd +(nStart - 1);
		END_IF
	ELSIF stItem.nCodeStartPos >= 0 AND stItem.nCodeLength > 0 THEN
		nStart := stItem.nCodeStartPos;
		nEnd := nStart + stItem.nCodeLength;
	ELSE
		nStart := 0;
		nEnd := 0;
	END_IF
	IF nStart > 0 AND nEnd > 0 THEN
		sItem := MID(sFullCode, nEnd - nStart, nStart);
	ELSE
		sItem := '';
	END_IF
ELSE
	sItem := '';
END_IF

F_CODE_GetItem := sItem;

END_FUNCTION

// ---- POUs/METS/Common LIB/04_CASE LIB/Case FBs/FB_CASE_ShiftPackerQueue.TcPOU
(* shifts specified group of cases from Packer layer 0 to Packer layer 1 *)
FUNCTION_BLOCK FB_CASE_ShiftPackerQueue
VAR_INPUT
	bExecute				: BOOL;			(* set TRUE to shift Case Queue *)
END_VAR
VAR_IN_OUT
	aPackerQueue 			: ARRAY [0..1] OF ST_CASE_InfeedQueue;	(* Outfeed Queue *)
END_VAR
VAR_OUTPUT
	bDone				: BOOL;			(* TRUE = complete *)
END_VAR
VAR
	fbExecute				: R_TRIG;
END_VAR

(* rising edge of bExecute *)
fbExecute(CLK:= bExecute);

(* move CaseData *)
IF fbExecute.Q = TRUE THEN

	(* shift specified*)
	MEMMOVE(ADR(aPackerQueue[1]), ADR(aPackerQueue[0]), SIZEOF(aPackerQueue[0]));
	(* clear data *)
	MEMSET(ADR(aPackerQueue[0]), 16#00, SIZEOF(aPackerQueue[0]));

	bDone := TRUE;

(* bExecute has been reset *)
ELSIF bExecute = FALSE THEN
	bDone := FALSE;
END_IF

END_FUNCTION_BLOCK

// ---- POUs/_Exclude/FB_CASE_FinaliseCaseData.TcPOU
(* move Outer data from sInfeedQueue to stCACData *)
FUNCTION_BLOCK FB_CASE_FinaliseCaseData
VAR_INPUT
	bExecute 			: BOOL;		(* set TRUE to move Outers *)
	stCTDateTime			: ST_SYSTEM_DateTime;
	strLocalOACPath		: STRING(255);	(* path to CaseTrace OAC folder *)
	strLocalOCVPath		: STRING(255);	(* path to CaseTrace OAC folder *)
	bUseInterimCodeForValidation	: BOOL;
END_VAR
VAR_IN_OUT
	stProductInstruction			: ST_PCM_Status;
	aOCVPackStatus			: ARRAY[1..cMAX_OUTER_STATUS_QUEUE] OF ST_OUTER_Status;	(* Outer status array *)
	aOuterStatus				: ARRAY[1..cMAX_OUTER_STATUS_QUEUE] OF ST_OUTER_Status;	(* Outer status array *)

	stCACData 				: ST_CAC_Data;	(* Case Queue *)
	stCACDataHMI			: ST_HMI_CAC_Data;

	stOuterRejectReasons			: ST_RejectReasonsForOuter;
	stCaseRejectReasons			: ST_RejectReasonsForCase;
	stCodeInfo_Pack				: ST_CodeInfo;
	stCodeInfo_Intermediate		: ST_CodeInfo;
	stCodeInfo_Outer				: ST_CodeInfo;
END_VAR
VAR_OUTPUT
	bDone 				: BOOL;		(* TRUE = move complete *)
	bBusy				: BOOL;
	bError				: BOOL;
	nErrorID 				: UDINT;
	bCACValid			: BOOL;
	bCACInvalid			: BOOL;
	strRejectCode		: STRING(255);
	bIsDuplicateOuterCodes:	BOOL;
	bIsDuplicatePackCodes:	BOOL;

	aDuplicatesOuters:			ARRAY[1..2] OF T_OUTER_Barcode;
	aDuplicatesPacks:			ARRAY[1..2] OF T_PACK_Barcode;

	nValidationIndex		: INT;
	nMasterListCounter		: INT;

	sCaseContent			: T_LongSTRING;
END_VAR
VAR
	fbExecute			: R_TRIG;
	eState				: E_CASE_STATE;
	eErrorState			: E_CASE_STATE;
	fbCaseContentValidation	: FB_CASE_ValidateCaseContent;

	nIndex					: T_PositiveINT;
	nIndexOuter: T_PositiveINT;
	nIndexPack: T_PositiveINT;

	bDoorReject: BOOL;
	sIntrimCode				: STRING(255);
	aAggregationCodes 			: ARRAY[1..2] OF T_PACK_Barcode;
	aOCVFileCodeName			: ARRAY[1..2] OF T_MaxString;
	strOACFile				: STRING(255);
	strOCVFile				: STRING(255);
	fbMoveFile				: FB_FILE_Move;
	nOACDeleteIndex			: INT;
	nOACFilesDeleted			: INT;
	nOCVFilesDeleted			: INT;
	nCaseContentLogIndex	: INT;
	sAppendedString		: STRING;
END_VAR

(* rising edge of bExecute *)
fbExecute(CLK:= bExecute);

CASE eState OF

	E_CASE_IDLE:

		(* validate stCACData *)
		IF fbExecute.Q THEN

			(* update outputs *)
			bDone 			:= FALSE;
			bBusy			:= TRUE;
			bError 			:= FALSE;
			nErrorID 		:= 0;

			(* clear outputs *)
			bCACValid 				:= FALSE;
			bCACInvalid 			:= FALSE;
			nValidationIndex 		:= 0;
			nMasterListCounter	 :=0;

			strRejectCode 	:= '';
			bDoorReject 	:= FALSE;
			(*IF stCACData.CaseRejectCode = stCaseRejectReasons.stDoorGuardReject.sMetsDisplayCode THEN
				bDoorReject := TRUE;
			ELSE
				bDoorReject := FALSE;
			END_IF*)
			(* populate case data *)
			(* date (YYYY-MM-DD) and time (hh:mm:ss) with offset to UTC *)
			stCACData.ProductionDate := F_StringWildcard('#YYYYMMDD#', stCTDateTime.sSystemTime);
			stCACData.ProductionTime := F_StringWildcard('#hhmmss#', stCTDateTime.sSystemTime);
			stCACData.ProductionTimeOffset := F_SYSTEM_SystemTimeOffsetToHHMM(stCTDateTime.nSystemTimeOffset);

			(* product and machine info *)
			stCACData.RetailSKU := stProductInstruction.sRetailSKU;    (*sCPIData.RetailSKU;*)
			stCACData.CasePacker.ProductionSite := stProductInstruction.sProductionSite; (*sCPIData.ProductionSite  ;*)
			stCACData.CasePacker.ProductionLine :=stProductInstruction.sProductionLine;  (*   sCPIData.ProductionLine;*)
			stCACData.CodingAndTrackingMode := stProductInstruction.nOpMode;  (*STRING_TO_INT(sCPIData.CodingAndTrackingMode);*)

			(* PassThrough, PrePrintedLabel or PrintApply mode active *)
			IF stCACData.CodingAndTrackingMode <= 6 THEN

				(* non-aggregated case, populate NumberOfOuters and CodingAndTrackingMode *)
				stCACData.NumberOfOuters := stProductInstruction.nOutersPerCase;

				stCACData.CaseRejectCode := 'OK';
				stCACData.CaseRejectID := 0;

				(* validation not required in these modes *)
				eState := E_CASE_DONE;

			(* CaseTrace or PackTrace mode *)
			ELSE
				FOR nIndex := 1 TO stProductInstruction.nOutersPerCase DO
					IF stCACData.Outer[nIndex].OuterMasterListRestored THEN
						nMasterListCounter := nMasterListCounter +1;
					END_IF
				END_FOR

				eState := E_CASE_VALIDATECAC;
			END_IF

		(* bExecute has been reset *)
		ELSIF bExecute = FALSE THEN

			bDone := FALSE;
			bBusy := FALSE;
			bError := FALSE;
			nErrorID := 0;
		END_IF


	(* validate CAC data *)
	E_CASE_VALIDATECAC:

		IF stCACData.CaseRejectCode = stCaseRejectReasons.stDoorGuardReject.sMetsDisplayCode THEN
			bDoorReject := TRUE;
		END_IF

		(* validate CAC *)
		fbCaseContentValidation(
			bExecute		:= TRUE,
			stCTDateTime	:= stCTDateTime,
			stCACData		:= stCACData,
			stProductInstruction := stProductInstruction,
			nSecquentionalCounter	:= gDevice.nDummySecquentionalCounter,
			stOuterCodeInfo	:= stCodeInfo_Outer,
			stOuterBarcodeDuplicate	:= stOuterRejectReasons.stOuterBarcodeDuplicate,
			stOuterDuplicatedPackCodesFound	:= stOuterRejectReasons.stOuterDuplicatedPackCodesFound,
			stCaseRejectReasons := stCaseRejectReasons,
			bIsDuplicateOuters=> bIsDuplicateOuterCodes,
			bIsDuplicatePacks=> bIsDuplicatePackCodes,
			aDuplicatesOuters=> aDuplicatesOuters,
			aDuplicatesPacks=> aDuplicatesPacks
		);

		(* validate CAC complete *)
		IF fbCaseContentValidation.bDone = TRUE THEN

			(* validate CAC completed OK *)
			IF fbCaseContentValidation.bError = TRUE THEN

				(* update status *)
				bError := TRUE;
				nErrorID := fbCaseContentValidation.nErrorID;
				eErrorState := eState;
			END_IF

			(* update RejectCode *)
			strRejectCode := stCACData.CaseRejectCode;
			nValidationIndex := stCACData.NumberOfOuters;

			IF bIsDuplicateOuterCodes OR bIsDuplicatePackCodes THEN
				nOACDeleteIndex	:= 1;
				MEMSET(ADR(aAggregationCodes), 16#00, SIZEOF(aAggregationCodes));
	
				eState :=  E_CASE_DELETEOACFILE;
			ELSE
				eState := E_CASE_DONE;
			END_IF

			(* close off fbValidateCAC *)
			fbCaseContentValidation(
				bExecute	:= FALSE,
				stCACData	:= stCACData,
				stProductInstruction := stProductInstruction,
				nSecquentionalCounter	:= gDevice.nDummySecquentionalCounter,
				stOuterCodeInfo	:= stCodeInfo_Outer,
				stOuterBarcodeDuplicate	:= stOuterRejectReasons.stOuterBarcodeDuplicate,
				stOuterDuplicatedPackCodesFound	:= stOuterRejectReasons.stOuterDuplicatedPackCodesFound,
				stCaseRejectReasons := stCaseRejectReasons
			);

		END_IF

(* delete OCV to error folder *)
	E_CASE_DELETEOACFILE:

		FOR nIndex := 1 TO cMAX_OUTER_STATUS_QUEUE DO
			IF aOuterStatus[nIndex].stOACData.Barcode =  aDuplicatesOuters[nOACDeleteIndex] AND aOuterStatus[nIndex].stOACData.Barcode <> '' THEN
				sIntrimCode := aOuterStatus[nIndex].stOACData.AggregationCodes[1];
				MEMSET(ADR(aOuterStatus[nIndex].stOACData), 16#00, SIZEOF(aOuterStatus[nIndex].stOACData));
				aOuterStatus[nIndex].nStatus.22 := TRUE;
				aOuterStatus[nIndex].stOACData.DataSource := 'REM';
				EXIT;
			END_IF
		END_FOR

		(* generate OAC file name and clear data for last OAC file *)

		strOACFile := F_CONCAT3('OAC_', F_OUTER_BarcodeToHex(aDuplicatesOuters[nOACDeleteIndex], stCodeInfo_Outer), '.xml');


		(* delete OCV file *)
		fbMoveFile(
				bExecute			:= TRUE,
				strPathSource		:= strLocalOACPath,
				strPathTarget		:= CONCAT(strLocalOACPath,'Error\' ),
				strFileName		:= strOACFile,
				tTimeout			:= T#1s
		);

		(* delete file complete *)
		IF fbMoveFile.bBusy = FALSE THEN

			(* delete  file completed OK *)
			IF fbMoveFile.bError = FALSE THEN

				(* update counter *)
				nOACFilesDeleted := nOACFilesDeleted + 1;

			(* delete command error or file not found *)
			ELSE

				bError := TRUE;
				nErrorID := fbMoveFile.nErrorID;
				eErrorState := eState;

			END_IF

			eState := E_CASE_DELETEOCV1FILE;

			(* close off fbDeleteOCVFile *)
			fbMoveFile(bExecute := FALSE);
		END_IF

	(* delete OCV to error folder *)
	E_CASE_DELETEOCV1FILE:

		FOR nIndex := 1 TO stProductInstruction.nOutersPerCase DO
			IF stCACData.Outer[nIndex].Barcode = aDuplicatesOuters[nOACDeleteIndex] THEN

				aAggregationCodes[1] := stCACData.Outer[nIndex].AggregationCodes[1];
			END_IF
		END_FOR

		IF aAggregationCodes[1] <> '' THEN

			FOR nIndex := 1 TO cMAX_OUTER_STATUS_QUEUE DO
				IF aOCVPackStatus[nIndex].stOACData.AggregationCodes[1] =  aAggregationCodes[1] THEN
					MEMSET(ADR(aOCVPackStatus[nIndex].stOACData), 16#00, SIZEOF(aOCVPackStatus[nIndex].stOACData));
					aOCVPackStatus[nIndex].nStatus.22 := TRUE;
					aOCVPackStatus[nIndex].stOACData.DataSource := 'REM';
					EXIT;
				END_IF
			END_FOR

			aOCVFileCodeName[1]	:=	F_CodeToHex(F_CODE_GetItem(aAggregationCodes[1] , eCodeAIType.SerialCode,
														SEL(bUseInterimCodeForValidation, stCodeInfo_Pack, stCodeInfo_Intermediate)));
			strOCVFile := F_CONCAT3('OCV_',aOCVFileCodeName[1], '.xml');
		END_IF

		(* delete OCV file *)
		fbMoveFile(
				bExecute			:= TRUE,
				strPathSource		:= strLocalOCVPath,
				strPathTarget		:= CONCAT(strLocalOCVPath,'Error\' ),
				strFileName		:= strOCVFile,
				tTimeout			:= T#1s
		);

		(* delete file complete *)
		IF fbMoveFile.bBusy = FALSE THEN

			(* delete  file completed OK *)
			IF fbMoveFile.bError = FALSE THEN

				(* update counter *)
				nOCVFilesDeleted := nOCVFilesDeleted + 1;

			(* delete command error or file not found *)
			ELSE

				bError := TRUE;
				nErrorID := fbMoveFile.nErrorID;
				eErrorState := eState;

			END_IF

			eState := E_CASE_DELETEOCV2FILE;

			(* close off fbDeleteOCVFile *)
			fbMoveFile(bExecute := FALSE);
		END_IF

	(* delete OCV to error folder *)
	E_CASE_DELETEOCV2FILE:

		FOR nIndex := 1 TO stProductInstruction.nOutersPerCase DO
			IF stCACData.Outer[nIndex].Barcode = aDuplicatesOuters[nOACDeleteIndex] THEN

				aAggregationCodes[2] := stCACData.Outer[nIndex].AggregationCodes[2];
				EXIT;
			END_IF
		END_FOR

		IF aAggregationCodes[2] <> '' THEN

			FOR nIndex := 1 TO cMAX_OUTER_STATUS_QUEUE DO
				IF aOCVPackStatus[nIndex].stOACData.AggregationCodes[2] =  aAggregationCodes[2] THEN
					MEMSET(ADR(aOCVPackStatus[nIndex].stOACData), 16#00, SIZEOF(aOCVPackStatus[nIndex].stOACData));
					aOCVPackStatus[nIndex].nStatus.22 := TRUE;
					aOCVPackStatus[nIndex].stOACData.DataSource := 'REM';
				END_IF
			END_FOR
			aOCVFileCodeName[2]	:=	F_CodeToHex(F_CODE_GetItem(aAggregationCodes[2] , eCodeAIType.SerialCode,   stCodeInfo_Pack)); (*no reason to have 2 diffrent intermediate codes*)
			strOCVFile := F_CONCAT3('OCV_',aOCVFileCodeName[2] , '.xml');
		END_IF


		(* delete OCV file *)
		fbMoveFile(
				bExecute			:= TRUE,
				strPathSource		:= strLocalOCVPath,
				strPathTarget		:= CONCAT(strLocalOCVPath,'Error\' ),
				strFileName		:= strOCVFile,
				tTimeout			:= T#1s
		);

		(* delete file complete *)
		IF fbMoveFile.bBusy = FALSE THEN

			(* delete  file completed OK *)
			IF fbMoveFile.bError = FALSE THEN

				(* update counter *)
				nOCVFilesDeleted := nOCVFilesDeleted + 1;

			(* delete command error or file not found *)
			ELSE

				bError := TRUE;
				nErrorID := fbMoveFile.nErrorID;
				eErrorState := eState;

			END_IF

			IF nOACDeleteIndex  <  2 THEN
				nOACDeleteIndex := nOACDeleteIndex +1;

				eState := E_CASE_DELETEOACFILE;
			ELSE
				eState := E_CASE_DONE;
			END_IF

			(* close off fbDeleteOCVFile *)
			fbMoveFile(bExecute := FALSE);
		END_IF

	(* complete *)
	E_CASE_DONE:

		IF bDoorReject THEN

			bError := TRUE;
			nErrorID := 20;
			eErrorState := eState;
			stCACData.CaseRejectCode := stCaseRejectReasons.stDoorGuardReject.sMetsDisplayCode;
			stCACData.CaseRejectID := stCaseRejectReasons.stDoorGuardReject.nRejectID;
		END_IF

(******************************************************************************************************************************************)

	(* clear HMI data *)
	MEMSET(ADR(stCACDataHMI), 16#00, SIZEOF(stCACDataHMI));

	(*copy data to stCaseQueueHMI[1]*)
	IF stCACData.CaseRejectCode = 'OK' THEN
		stCACDataHMI.sBarcode:= F_CONCAT3(stCACData.Barcode,'(999)','1');
	ELSE
		stCACDataHMI.sBarcode:= F_CONCAT3(stCACData.Barcode,'(999)','0');
	END_IF

	stCACDataHMI.nNumberOfOuters 	:= stCACData.NumberOfOuters;
	stCACDataHMI.nNumberOfPacks 		:= stCACData.Outer[1].NumberOfPacks;

	FOR nIndexOuter:=1 TO MIN(stCACData.NumberOfOuters, cMAX_OUTERS_PER_CASE) DO
		IF stCACData.Outer[nIndexOuter].OuterRejectCode = 'OK' THEN
			stCACDataHMI.aOuter[nIndexOuter].sBarcode:= F_CONCAT3(stCACData.Outer[nIndexOuter].Barcode,'(999)','1');
		ELSE
			stCACDataHMI.aOuter[nIndexOuter].sBarcode:= F_CONCAT3(stCACData.Outer[nIndexOuter].Barcode,'(999)','0');
		END_IF

		FOR nIndexPack:=1 TO MIN(stCACData.Outer[nIndexOuter].NumberOfPacks, cMAX_PACKS_PER_OUTER) DO
			IF stCACData.Outer[nIndexOuter].PackRejectCode[nIndexPack] = 'OK' THEN
				stCACDataHMI.aOuter[nIndexOuter].aPackCode[nIndexPack]:= F_CONCAT3(stCACData.Outer[nIndexOuter].PackCode[nIndexPack],'(999)','1');
			ELSE
				stCACDataHMI.aOuter[nIndexOuter].aPackCode[nIndexPack]:= F_CONCAT3(stCACData.Outer[nIndexOuter].PackCode[nIndexPack],'(999)','0');
			END_IF

		END_FOR
	END_FOR

(******************************************************************************************************************************************)
		sAppendedString	:= '';
		sCaseContent 	:= '';
		
		sCaseContent := F_CONCAT3(' [', INT_TO_STRING(stCACData.NumberOfOuters),']:');
		FOR nCaseContentLogIndex := 1 TO MIN(stCACData.NumberOfOuters ,cMAX_OUTERS_PER_CASE) BY 1 DO
			//sCaseContent :=F_LongCONCAT(sCaseContent, '   ');
			//sCaseContent := F_LongCONCAT(sCaseContent, RIGHT(F_CODE_GetItem(stCACData.Outer[nCaseContentLogIndex].Barcode, eCodeAIType.SerialCode,  stCodeInfo_Outer),7));
		
			CONCAT2(ADR(sCaseContent), ADR('   '), ADR(sCaseContent), SIZEOF(sCaseContent));
		
			sAppendedString := RIGHT(F_CODE_GetItem(stCACData.Outer[nCaseContentLogIndex].Barcode, eCodeAIType.SerialCode,  stCodeInfo_Outer),7);
			CONCAT2(ADR(sCaseContent), ADR(sAppendedString), ADR(sCaseContent), SIZEOF(sCaseContent));
		END_FOR

		(* no error occured *)
		IF bError = FALSE THEN

			(* CAC data is valid *)
			bCACValid := TRUE;
			bCACInvalid := FALSE;

		(* invalid CAC *)
		ELSE

			(* CAC data is invalid *)
			bCACValid := FALSE;
			bCACInvalid := TRUE;
		END_IF



		(* update outputs *)
		bBusy := FALSE;
		bDone := TRUE;

		eState := E_CASE_IDLE;


(* unknown state *)
ELSE

	eState := E_CASE_IDLE;
END_CASE

END_FUNCTION_BLOCK

// ---- POUs/_Exclude/FB_CASE_ValidateCaseContent.TcPOU
(* move Outer data from sInfeedQueue to stCACData *)
FUNCTION_BLOCK FB_CASE_ValidateCaseContent
VAR_INPUT
	bExecute 						: BOOL;
	stCTDateTime					: ST_SYSTEM_DateTime;	(* CaseTrace date/time structure *)
END_VAR
VAR_IN_OUT
	stCACData 						: ST_CAC_Data;
	stProductInstruction				: ST_PCM_Status;
	nSecquentionalCounter			: UDINT;
	stOuterCodeInfo						: ST_CodeInfo;
	stOuterBarcodeDuplicate			: ST_RejectItems;
	stOuterDuplicatedPackCodesFound	: ST_RejectItems;
	stCaseRejectReasons			: ST_RejectReasonsForCase;
END_VAR
VAR_OUTPUT
	bDone 						: BOOL;
	bBusy						: BOOL;
	bError						: BOOL;
	nErrorID 						: UDINT;
	bCACValid					: BOOL;
	strRejectCode					: STRING(255);
	bIsDuplicateOuters		: BOOL;
	bIsDuplicatePacks		: BOOL;
	aDuplicatesOuters					: ARRAY[1..2] OF T_OUTER_Barcode;
	aDuplicatesPacks					: ARRAY[1..2] OF T_PACK_Barcode;

END_VAR
VAR
	fbExecute						: R_TRIG;
	eState						: E_CAC_STATE;
	eErrorState					: E_CAC_STATE;

	(*nIndex						: INT;*)

	bValQtyOver				: BOOL;

	(*fbValidateCaseLabel				: FB_CODE_ValidateExplicitCode;*)
	nOutGTIN						: INT;
	nOutBand						: INT;
	nRetailSKU					: INT;
	nSerialCode					: INT;
	nTotalInvalide					: INT;

	fbValidateOuter				: FB_CODE_ValidateExplicitCode;
	nValidOACData					: INT;

	(*fbValidatePack					: FB_CODE_ValidateExplicitCode;*)
	nOuterIndex					: INT;
	nPackIndex					: INT;
	nValidPackData					: INT;
	nIndex2: T_PositiveINT;
	nIndex3: T_PositiveINT;

	aStatusErrorVal					: ARRAY[0..10] OF STRING(10);
	aRejectCodePointer     		   	: ARRAY[0..10] OF STRING(10);

	aOuterBarcodes				: ARRAY[1..cMAX_OUTERS_PER_CASE] OF T_OUTER_Barcode;
	aPackBarcodes					: ARRAY[1..cMAX_PACK_PER_CASE] OF ST_PACK_DuplicatesCheck;

	nIndex4: T_PositiveINT;
	nIndex5: T_PositiveINT;
	nIndex6: T_PositiveINT :=1;
	nOuterCheckedIndex: T_PositiveINT;
	nOuterIndexDupCheck : T_PositiveINT;
	sCurrentOuterCheck	:T_OUTER_Barcode;
	nPackCheckedIndex: T_PositiveINT;
	nPackIndexDupCheck : T_PositiveINT;
	sCurrentPackCheck	:T_PACK_Barcode;
	nDuplicateOuter1_Position: T_PositiveINT;
	nDuplicateOuter2_Position: T_PositiveINT;
	nDuplicatePack1_Position: T_PositiveINT;
	nDuplicatePack2_Position: T_PositiveINT;
END_VAR

(* rising edge of bExecute *)
fbExecute(CLK:= bExecute);

CASE eState OF

	E_CAC_IDLE:

		(* validate stCACData *)
		IF fbExecute.Q THEN

			(* update outputs *)
			bDone := FALSE;
			bBusy := TRUE;
			bError := FALSE;
			nErrorID := 0;
			bIsDuplicateOuters:= FALSE;
			bIsDuplicatePacks:= FALSE;
			MEMSET(ADR(aDuplicatesOuters),16#00,SIZEOF(aDuplicatesOuters));
			MEMSET(ADR(aDuplicatesPacks),16#00,SIZEOF(aDuplicatesPacks));

			MEMSET(ADR(aStatusErrorVal), 16#00, SIZEOF(aStatusErrorVal));
			MEMSET(ADR(aRejectCodePointer), 16#00, SIZEOF(aRejectCodePointer));

			MEMSET(ADR(aOuterBarcodes),16#00,SIZEOF(aOuterBarcodes));
			MEMSET(ADR(aPackBarcodes),16#00,SIZEOF(aPackBarcodes));

			nIndex6 := 1;
			nDuplicateOuter1_Position :=0;
			nDuplicateOuter2_Position:=0;
			nDuplicatePack1_Position:=0;
			nDuplicatePack2_Position:=0;
			sCurrentOuterCheck := '';
			sCurrentPackCheck := '';

			(* clear outputs *)
			bCACValid := FALSE;
			strRejectCode := '';

			eState := E_CAC_VALIDATECASE;

		(* bExecute has been reset *)
		ELSIF bExecute = FALSE THEN

			(* clear outputs *)
			bDone := FALSE;
			bBusy := FALSE;
			bError := FALSE;
			(*nErrorID := 0;*)
		END_IF


	(* validate Case data *)
	E_CAC_VALIDATECASE:

		(* Create a strucuture of Outer Barcodes to Duplicates Check *)
		FOR nIndex4 :=1 TO stProductInstruction.nOutersPerCase DO

			IF nIndex4 <= cMAX_OUTERS_PER_CASE THEN
				aOuterBarcodes[nIndex4] := stCACData.Outer[nIndex4].Barcode;

				IF stCACData.Outer[nIndex4].OuterCodeStatus.5 AND stCACData.NumberOfOuters = stProductInstruction.nOutersPerCase  THEN
					stCACData.NumberOfOuters := -3;		//b5		Outer Code - Val Index error found
				END_IF
			END_IF

			(* Create a strucuture of Pack Codes for Duplicates Check *)
			FOR nIndex5 :=1 TO stProductInstruction.nPacksPerOuter  DO

				IF nIndex6 <= cMAX_PACK_PER_CASE THEN
					nIndex6 := (nIndex4 * stProductInstruction.nPacksPerOuter)  - stProductInstruction.nPacksPerOuter + nIndex5;
	
					aPackBarcodes[nIndex6  ].sPackcode := stCACData.Outer[nIndex4].PackCode[nIndex5];
					aPackbarcodes[nIndex6].nPackRejectID := stCACData.Outer[nIndex4].PackRejectID[nIndex5];
					aPackBarcodes[nIndex6].nOuterIndex := nIndex4;
					aPackBarcodes[nIndex6].nPackIndex := nIndex5;
				END_IF

			END_FOR
		END_FOR

		(* Outers in Case is correct *)
		IF stCACData.NumberOfOuters = stProductInstruction.nOutersPerCase THEN

			(* Outer aggregation enabled *)
			IF stCACData.CodingAndTrackingMode >= 7 THEN

				eState := E_CAC_VALIDATEOUTER;

			(* OAC data disabled *)
			ELSE

				eState := E_CAC_DONE;
			END_IF

		(* invalid Case *)
		ELSE

			(* update status *)
			bError := TRUE;
			eErrorState := eState;

			(* no validation code read *)
			IF stCACData.NumberOfOuters = -1 THEN

				(* error code *)
				nErrorID := 11;

				(* reset nNumberOfOuters to 0 and generate reject string *)
				stCACData.NumberOfOuters := 0;

				stCACData.CaseRejectCode :=  stCaseRejectReasons.stCaseNoCaseData.sMetsDisplayCode;
				stCACData.CaseRejectID := stCaseRejectReasons.stCaseNoCaseData.nRejectID;
			(* validation code not found in sInfeedQueue *)
			ELSIF stCACData.NumberOfOuters = -2 THEN

				(* error code *)
				nErrorID := 12;

				(* reset nNumberOfOuters to 0 and generate reject string *)
				stCACData.NumberOfOuters := 0;

				aStatusErrorVal[0] := 	INT_TO_STRING(stCACData.NumberOfOuters);
				aRejectCodePointer[0] := 'nn';

				stCACData.CaseRejectCode 	:=	F_CODE_AssignValToStringWithPrefix(stCaseRejectReasons.stValError.sMetsDisplayCode, aStatusErrorVal, aRejectCodePointer, 3, '0');
				stCACData.CaseRejectID := stCaseRejectReasons.stValError.nRejectID;

				(*eState := E_CAC_DONE;*)

			ELSIF stCACData.NumberOfOuters = -3 THEN


				(* error code *)
				nErrorID := 13;

				(* reset nNumberOfOuters to 0 and generate reject string *)
				stCACData.NumberOfOuters := stProductInstruction.nOutersPerCase;

				aStatusErrorVal[0] := 	INT_TO_STRING(stCACData.NumberOfOuters);
				aRejectCodePointer[0] := 'nn';

				stCACData.CaseRejectCode 	:=	F_CODE_AssignValToStringWithPrefix(stCaseRejectReasons.stValError.sMetsDisplayCode, aStatusErrorVal, aRejectCodePointer, 3, '0');
				stCACData.CaseRejectID := stCaseRejectReasons.stValError.nRejectID;

				(*eState := E_CAC_DONE;*)

			(* incorrect number of Outers *)
			ELSE

				(* generate reject string *)

				aStatusErrorVal[0] := 	INT_TO_STRING(stCACData.NumberOfOuters);
				aRejectCodePointer[0] := 'nn';

				stCACData.CaseRejectCode 	:=	F_CODE_AssignValToStringWithPrefix(stCaseRejectReasons.stValError.sMetsDisplayCode, aStatusErrorVal, aRejectCodePointer, 3, '0');
				stCACData.CaseRejectID := stCaseRejectReasons.stValError.nRejectID;

				(* >=1 Outer(s) missed by Infeed camera *)
				IF stCACData.NumberOfOuters < stProductInstruction.nOutersPerCase THEN

					(* error code *)
					nErrorID := 14;

				(* >=1 Outer(s) physically removed from Infeed queue *)
				ELSE

					(* error code *)
					nErrorID := 15;
				END_IF
			END_IF

			eState := E_CAC_DONE;
		END_IF

	(* validate RetailSKU for each Outer *)
	E_CAC_VALIDATEOUTER:

		(* initialise counters *)
		nOutGTIN		:= 0;
		nOutBand		:= 0;
		nRetailSKU 	:= 0;
		nSerialCode 	:= 0;
		nTotalInvalide	:= 0;

		(* for each Outer *)
		FOR nOuterIndex := 1 TO stCACData.NumberOfOuters DO

			fbValidateOuter(	sFullCode := stCACData.Outer[nOuterIndex].Barcode,
							stCodeInfo := stOuterCodeInfo,
							stProductInstruction := stProductInstruction);

			IF fbValidateOuter.bGtinOK  THEN

				(* Outer has valid GTIN *)
				nOutGTIN := nOutGTIN + 1;
			END_IF

			IF fbValidateOuter.bBrandOK  THEN

				(* Outer has valid GTIN *)
				nOutBand := nOutBand + 1;
			END_IF


			IF fbValidateOuter.bSerialCodeOK  THEN

				(* Outer has valid SerialCode *)
				nSerialCode := nSerialCode + 1;
			END_IF

			IF fbValidateOuter.bRskuOK  THEN

				(* Outer has valid RetailSKU *)
				nRetailSKU := nRetailSKU + 1;
			END_IF

			IF fbValidateOuter.bValidationOK THEN

				(* Total number of invalide outers - whatever reaso*)
				nTotalInvalide := nTotalInvalide +1;
			END_IF
		END_FOR


		(* all Outers have valid GTIN *)
		IF  nOutGTIN = stProductInstruction.nOutersPerCase THEN
			(* all Outers have valid Brand *)
			IF  nOutBand = stProductInstruction.nOutersPerCase THEN
				(* all Outers have valid RetailSKU *)
				IF  nRetailSKU = stProductInstruction.nOutersPerCase  THEN
					(* all Outers have valid SerialCode *)
					IF  nSerialCode = stProductInstruction.nOutersPerCase THEN
						(*If total invalide Outers inside a case*)
						IF  nTotalInvalide = stProductInstruction.nOutersPerCase THEN
	
							eState := E_CAC_VALIDATEOAC;
	
						ELSE
							(* RejectCode *)
							bError := TRUE;
							nErrorID := 16;
							eErrorState := eState;
					
							aStatusErrorVal[0] 		:=  INT_TO_STRING(stCACData.NumberOfOuters - nTotalInvalide);
							aRejectCodePointer[0] 	:= 'nn';
						
							stCACData.CaseRejectCode 	:=	F_CODE_AssignValToStringWithPrefix(stCaseRejectReasons.stINVError.sMetsDisplayCode, aStatusErrorVal, aRejectCodePointer, 2, '0');
							stCACData.CaseRejectID 		:= stCaseRejectReasons.stINVError.nRejectID;
							eState := E_CAC_DONE;

						END_IF
					(* 1 or more Outers have incorrect SerialCode *)
					ELSE
		
						(* RejectCode *)
						bError := TRUE;
						nErrorID := 17;
						eErrorState := eState;
	
						(* generate reject string *)
	
						aStatusErrorVal[0] 		:=  INT_TO_STRING(stCACData.NumberOfOuters - nSerialCode);
						aRejectCodePointer[0] 	:= 'nn';
	
						stCACData.CaseRejectCode 	:=	F_CODE_AssignValToStringWithPrefix(stCaseRejectReasons.stOuterSerialError.sMetsDisplayCode, aStatusErrorVal, aRejectCodePointer, 2, '0');
						stCACData.CaseRejectID := stCaseRejectReasons.stOuterSerialError.nRejectID;
						(*eState := E_CAC_DONEAS;*) (*AS Mod This original code line changed to do OAC check even if there are SERC errors*)
						eState := E_CAC_DONE;
	
					END_IF
	
				(* 1 or more Outers with invalid RetailSKU *)
				ELSE
		
					(* RejectCode *)
					bError := TRUE;
					nErrorID := 18;
					eErrorState := eState;
		
					(* generate reject string *)
	
					aStatusErrorVal[0] 		:=  INT_TO_STRING(stCACData.NumberOfOuters - nRetailSKU);
					aRejectCodePointer[0] 	:= 'nn';
		
					stCACData.CaseRejectCode 	:=	F_CODE_AssignValToStringWithPrefix(stCaseRejectReasons.stOuterRSKUError.sMetsDisplayCode, aStatusErrorVal, aRejectCodePointer, 2, '0');
					stCACData.CaseRejectID := stCaseRejectReasons.stOuterRSKUError.nRejectID;
					eState := E_CAC_DONE;
	
				END_IF
			ELSE
				(* RejectCode *)
				bError := TRUE;
				nErrorID := 19;
				eErrorState := eState;
	
				(* generate reject string *)

				aStatusErrorVal[0] 		:=  INT_TO_STRING(stCACData.NumberOfOuters - nOutBand);
				aRejectCodePointer[0] 	:= 'nn';
	
				stCACData.CaseRejectCode 	:=	F_CODE_AssignValToStringWithPrefix(stCaseRejectReasons.stOuterBrandError.sMetsDisplayCode, aStatusErrorVal, aRejectCodePointer, 2, '0');
				stCACData.CaseRejectID := stCaseRejectReasons.stOuterBrandError.nRejectID;
				eState := E_CAC_DONE;
			END_IF
		ELSE
		(* RejectCode *)
			bError := TRUE;
			nErrorID := 20;
			eErrorState := eState;

			(* generate reject string *)

			aStatusErrorVal[0] 		:=  INT_TO_STRING(stCACData.NumberOfOuters - nOutGTIN);
			aRejectCodePointer[0] 	:= 'nn';

			stCACData.CaseRejectCode 	:=	F_CODE_AssignValToStringWithPrefix(stCaseRejectReasons.stOuterGTINError.sMetsDisplayCode, aStatusErrorVal, aRejectCodePointer, 2, '0');
			stCACData.CaseRejectID := stCaseRejectReasons.stOuterGTINError.nRejectID;
			eState := E_CAC_DONE;

		END_IF

(* check OAC data was loaded *)
	E_CAC_VALIDATEOAC:

		(* initialise counter *)
		nValidOACData := 0;

		(* for each Outer *)
		FOR nOuterIndex := 1 TO stCACData.NumberOfOuters DO

			IF stCACData.CodingAndTrackingMode = 7 THEN
				(* OAC mode >= CAC mode, OAC data will contain all data required for CAC mode *)
				IF  stCACData.Outer[nOuterIndex].DataSource <>  'NO_R' AND stCACData.Outer[nOuterIndex].CodingAndTrackingMode = stCACData.CodingAndTrackingMode  THEN
					(* count Outers with valid OAC data *)
					nValidOACData := nValidOACData + 1;
				END_IF
			ELSIF stCACData.CodingAndTrackingMode = 11 THEN
			(* CAC mode -> OAC data will contain all data required for CAC mode *)
				IF stCACData.Outer[nOuterIndex].DataSource <>  'NO_R'  AND stCACData.Outer[nOuterIndex].OuterRejectCode = 'OK'  THEN
					(* count Outers with valid OAC data *)
					nValidOACData := nValidOACData + 1;
				END_IF
			END_IF
		END_FOR

		(* all Outers with valid OAC data *)
		IF (nValidOACData *100 ) / stProductInstruction.nOutersPerCase   >=  stProductInstruction.nCaseAcceptanceLevelOuters THEN


			FOR nOuterIndex := 1 TO stCACData.NumberOfOuters DO

				IF stCACData.CodingAndTrackingMode >= 7 THEN
					(* CAC mode -> OAC data will contain all data required for CAC mode *)
						IF stCACData.Outer[nOuterIndex].DataSource =  'NO_R'  THEN

							stCACData.Outer[nOuterIndex].ProductionDate := F_StringWildcard('#YYYYMMDD#', stCTDateTime.sSystemTime);
							stCACData.Outer[nOuterIndex].ProductionTime := F_StringWildcard('#hhmmss#', stCTDateTime.sSystemTime);
							stCACData.Outer[nOuterIndex].ProductionTimeOffset := F_SYSTEM_SystemTimeOffsetToHHMM(stCTDateTime.nSystemTimeOffset);
		
							stCACData.Outer[nOuterIndex].OuterTimeStamp :=F_SYSTEM_SystemTimeAsISO8601(stCTDateTime.sSystemTime, stCTDateTime.sUTCTimeZoneOffset );
							stCACData.Outer[nOuterIndex].RetailSKU := stProductInstruction.sRetailSKU;
							stCACData.Outer[nOuterIndex].OuterMachine.ProductionSite :=  stProductInstruction.sProductionSite;
							stCACData.Outer[nOuterIndex].OuterMachine.ProductionLine := stProductInstruction.sProductionLine;
							stCACData.Outer[nOuterIndex].BatchNumber := stProductInstruction.sBatchNumber;
							stCACData.Outer[nOuterIndex].CodingAndTrackingMode := stProductInstruction.nOpMode;

							stCACData.Outer[nOuterIndex].NumberOfPacks	:=   stProductInstruction.nPacksPerOuter;
							stCACData.Outer[nOuterIndex].AcceptanceLevel	:= 	stProductInstruction.nAcceptanceLevel;

							stCACData.Outer[nOuterIndex].OuterRejectCode := 'OK';
							stCACData.Outer[nOuterIndex].OuterRejectID := 0;
							stCACData.Outer[nOuterIndex].DataSource :=  '3DC';

						ELSIF stCACData.Outer[nOuterIndex].DataSource <>  'NO_R'  AND stCACData.Outer[nOuterIndex].OuterRejectCode <> 'OK' THEN

							stCACData.Outer[nOuterIndex].OuterRejectCode := 'OK';
							stCACData.Outer[nOuterIndex].OuterRejectID := 0;
							stCACData.Outer[nOuterIndex].DataSource :=  '3DCR';
						END_IF
				END_IF
			END_FOR

			eState := E_CAC_CHECKOUTERDUPLICATES;

		(* 1 or more Outers with missing OAC data *)
		ELSE

			(* update status *)
			bError := TRUE;
			nErrorID := 21;
			eErrorState := eState;

			(* generate reject string *)

			aStatusErrorVal[0] := 	INT_TO_STRING(stCACData.NumberOfOuters - nValidOACData);
			aRejectCodePointer[0] := 'nn';

			stCACData.CaseRejectCode 	:=	F_CODE_AssignValToStringWithPrefix(stCaseRejectReasons.stOACError.sMetsDisplayCode, aStatusErrorVal, aRejectCodePointer, 3, '0');
			stCACData.CaseRejectID := stCaseRejectReasons.stOACError.nRejectID;

			eState := E_CAC_DONE;
		END_IF


	(* Check Outer for Duplicate Outer Labels*)
	E_CAC_CHECKOUTERDUPLICATES:

		FOR nOuterCheckedIndex := 1 TO MIN(stProductInstruction.nOutersPerCase,cMAX_OUTERS_PER_CASE) BY 1 DO
			sCurrentOuterCheck := aOuterBarcodes[nOuterCheckedIndex];
			(*Against every other outer ....*)
			FOR nOuterIndexDupCheck := nOuterCheckedIndex  TO  MIN(stProductInstruction.nOutersPerCase,cMAX_OUTERS_PER_CASE)  BY 1 DO
				IF sCurrentOuterCheck = aOuterBarcodes[nOuterIndexDupCheck]
					AND nOuterCheckedIndex <> nOuterIndexDupCheck
					AND sCurrentOuterCheck <> '' THEN

					bIsDuplicateOuters := TRUE;
					nDuplicateOuter1_Position := nOuterCheckedIndex;
					nDuplicateOuter2_Position := nOuterIndexDupCheck;
					EXIT;
				END_IF
				IF bIsDuplicateOuters THEN
					EXIT;
				END_IF
			END_FOR
			IF bIsDuplicateOuters THEN
				EXIT;
			END_IF
		END_FOR

		IF bIsDuplicateOuters THEN
			aStatusErrorVal[0] := 	INT_TO_STRING(nDuplicateOuter1_Position);
			aStatusErrorVal[1] := 	INT_TO_STRING(nDuplicateOuter2_Position);
			aRejectCodePointer[0] := 'n1';
			aRejectCodePointer[1] := 'n2';
			stCACData.CaseRejectCode 	:=	F_CODE_AssignValToStringWithPrefix(stCaseRejectReasons.stDUPError.sMetsDisplayCode, aStatusErrorVal, aRejectCodePointer, 2, '0');
			stCACData.CaseRejectID	:= 	stCaseRejectReasons.stDUPError.nRejectID;


			stCACData.Outer[nDuplicateOuter1_Position].OuterRejectCode 	:=	stOuterBarcodeDuplicate.sMetsDisplayCode;
			stCACData.Outer[nDuplicateOuter1_Position].OuterRejectID		:=	stOuterBarcodeDuplicate.nRejectID;

			stCACData.Outer[nDuplicateOuter2_Position].OuterRejectCode 	:=	stOuterBarcodeDuplicate.sMetsDisplayCode;
			stCACData.Outer[nDuplicateOuter2_Position].OuterRejectID		:=	stOuterBarcodeDuplicate.nRejectID;

			aDuplicatesOuters[1] := sCurrentOuterCheck;
			aDuplicatesOuters[2] := aOuterBarcodes[nOuterIndexDupCheck];

			(* update status *)
			bError := TRUE;
			nErrorID := 22;
			eErrorState := eState;

			eState := E_CAC_DONE;
		ELSE
			IF stCACData.CodingAndTrackingMode = 11 THEN

				eState := E_CAC_VALIDATEPACK;
			(* PackCode data disabled *)
			ELSE

			eState := E_CAC_DONE;
			END_IF
		END_IF

	(* check that PackCode data is included with OAC data *)
	E_CAC_VALIDATEPACK:

		(* initialise counter *)
		nValidPackData := 0;

		(* for each Outer *)
		FOR nOuterIndex := 1 TO stCACData.NumberOfOuters DO

			(* count Outers with PackCode data - assume- outer reject station working fine and only good outers in case, NumberOfLinkedPacks= good pack  *)
			nValidPackData := nValidPackData + stCACData.Outer[nOuterIndex].NumberOfLinkedPacks ;

			FOR nPackIndex := 1 TO stCACData.Outer[nOuterIndex].NumberOfPacks DO

				IF stCACData.Outer[nOuterIndex].PackCodeStatus[nPackIndex].1
					AND stCACData.Outer[nOuterIndex].PackCodeStatus[nPackIndex].2
					AND stCACData.Outer[nOuterIndex].PackCodeStatus[nPackIndex].3	THEN

					nValidPackData := -1;
					EXIT;
				END_IF
			END_FOR

			IF nValidPackData = -1 THEN
				EXIT;
			END_IF

		END_FOR

		(* Outers with PackCode data is correct *)
		IF (nValidPackData *100 ) /  stProductInstruction.nPacksPerCase  >=   stProductInstruction.nCaseAcceptanceLevelPacks   THEN

			FOR nOuterIndex := 1 TO stCACData.NumberOfOuters DO

				IF stCACData.Outer[nOuterIndex].NumberOfLinkedPacks = 0 THEN
					stCACData.Outer[nOuterIndex].PackTimeStamp := F_SYSTEM_SystemTimeAsISO8601(stCTDateTime.sSystemTime, stCTDateTime.sUTCTimeZoneOffset );
				END_IF

				FOR nPackIndex := 1 TO stCACData.Outer[nOuterIndex].NumberOfPacks DO
					(*Tolerance do not modify NumberOfLinkedPacks per outer*) (*later, repalce with PackCodeStatus.0*)
					IF  stCACData.Outer[nOuterIndex].PackCode[nPackIndex] = '' THEN

						stCACData.Outer[nOuterIndex].PackCode[nPackIndex] := F_CODE_BATSerializator(stCTDateTime, ePack, TRUE, stProductInstruction, nSecquentionalCounter);
						(* change reject reason to adjust for tolerance *)
						(*additional bit passing to CAC*)
						stCACData.Outer[nOuterIndex].PackCodeStatus[nPackIndex]:=
														F_FiltredSetBitState16(TRUE, 'LOW', 4, TRUE, stCACData.Outer[nOuterIndex].PackCodeStatus[nPackIndex]);

						stCACData.Outer[nOuterIndex].PackRejectCode[nPackIndex]  := 'OK';
						stCACData.Outer[nOuterIndex].PackRejectID[nPackIndex]		:= 0;
					END_IF
				END_FOR

				stCACData.Outer[nOuterIndex].NumberOfLinkedPacks := stCACData.Outer[nOuterIndex].NumberOfPacks;

			END_FOR

			eState := E_CAC_CHECKPACKDUPLICATES;

		ELSIF nValidPackData = -1 THEN

			(* RejectCode *)
			bError := TRUE;
			nErrorID := 23;
			eErrorState := eState;
	
			aStatusErrorVal[0] 		:=  'PK';
			aRejectCodePointer[0] 	:= 'nn';

			stCACData.CaseRejectCode 	:=	F_CODE_AssignValToStringWithPrefix(stCaseRejectReasons.stINVError.sMetsDisplayCode, aStatusErrorVal, aRejectCodePointer, 2, '0');
			stCACData.CaseRejectID 		:= stCaseRejectReasons.stINVError.nRejectID;

			eState := E_CAC_DONE;


		(* 1 or more Outers has no PackCode data *)
		ELSE

			(* update status *)
			bError := TRUE;
			nErrorID := 24;
			eErrorState := eState;

			(* generate reject string *)			(* generate reject string *)
			(*stCACData.RejectCode := F_CONCAT3('XXXPACK', F_StringAddPrefix(INT_TO_STRING(stCACData.NumberOfOuters - nValidPackData), 2, '0'), 'XXX');*)

			aStatusErrorVal[0] := 	INT_TO_STRING(stProductInstruction.nPacksPerCase - nValidPackData);
			aRejectCodePointer[0] := 'nn';

			stCACData.CaseRejectCode 	:=	F_CODE_AssignValToStringWithPrefix(stCaseRejectReasons.stPackNotLinedError.sMetsDisplayCode, aStatusErrorVal, aRejectCodePointer, 3, '0');
			stCACData.CaseRejectID := stCaseRejectReasons.stPackNotLinedError.nRejectID;

			eState := E_CAC_DONE;
		END_IF

	E_CAC_CHECKPACKDUPLICATES:
	(* Check whole Case for Duplicate Packs*)
		FOR nPackCheckedIndex := 1 TO MIN(stProductInstruction.nPacksPerCase, cMAX_PACK_PER_CASE) BY 1 DO
			sCurrentPackCheck := aPackBarcodes[nPackCheckedIndex].sPackcode;
			(*Against every other Pack ....*)
			FOR nPackIndexDupCheck := nPackCheckedIndex  TO MIN(stProductInstruction.nPacksPerCase, cMAX_PACK_PER_CASE) BY 1 DO
				IF sCurrentPackCheck = aPackBarcodes[nPackIndexDupCheck].sPackcode
					AND sCurrentPackCheck <> ''
					AND nPackCheckedIndex <> nPackIndexDupCheck
					AND aPackBarcodes[nPackCheckedIndex].nPackRejectID <> 107
					AND aPackBarcodes[nPackIndexDupCheck].nPackRejectID <> 107  THEN

						bIsDuplicatePacks := TRUE;
						nDuplicateOuter1_Position := aPackBarcodes[nPackCheckedIndex].nOuterIndex;
						nDuplicateOuter2_Position :=  aPackBarcodes[nPackIndexDupCheck].nOuterIndex;
						nDuplicatePack1_Position := aPackBarcodes[nPackCheckedIndex].nPackIndex;
						nDuplicatePack2_Position := aPackBarcodes[nPackIndexDupCheck].nPackIndex;
						EXIT;
				END_IF
				IF bIsDuplicatePacks THEN
					EXIT;
				END_IF
			END_FOR
			IF bIsDuplicatePacks THEN
				EXIT;
			END_IF
		END_FOR

		IF bIsDuplicatePacks THEN
			aStatusErrorVal[0] := 	F_CONCAT4(INT_TO_STRING(nDuplicateOuter1_Position),'(', INT_TO_STRING(nDuplicatePack1_Position),')');
			aStatusErrorVal[1] := 	F_CONCAT4(INT_TO_STRING(nDuplicateOuter2_Position),'(', INT_TO_STRING(nDuplicatePack2_Position),')');
	
			aRejectCodePointer[0] := 'n1';
			aRejectCodePointer[1] := 'n2';
	
			stCACData.CaseRejectCode 	:=	F_CODE_AssignValToStringWithPrefix(stCaseRejectReasons.stDUPError.sMetsDisplayCode, aStatusErrorVal, aRejectCodePointer, 2, '0');
			stCACData.CaseRejectID		:= stCaseRejectReasons.stDUPError.nRejectID;
	

			stCACData.Outer[nDuplicateOuter1_Position].OuterRejectCode 	:=	stOuterBarcodeDuplicate.sMetsDisplayCode;
			stCACData.Outer[nDuplicateOuter1_Position].OuterRejectID		:=	stOuterBarcodeDuplicate.nRejectID;
	
			stCACData.Outer[nDuplicateOuter2_Position].OuterRejectCode 	:=	stOuterBarcodeDuplicate.sMetsDisplayCode;
			stCACData.Outer[nDuplicateOuter2_Position].OuterRejectID		:=	stOuterBarcodeDuplicate.nRejectID;
	
			aDuplicatesOuters[1] := aOuterBarcodes[nDuplicateOuter1_Position];
			aDuplicatesOuters[2] := aOuterBarcodes[nDuplicateOuter2_Position];
			aDuplicatesPacks[1] := sCurrentPackCheck;
			aDuplicatesPacks[2] := aPackBarcodes[nPackIndexDupCheck].sPackcode;

			(* update status *)
			bError := TRUE;
			nErrorID := 25;
			eErrorState := eState;
		END_IF
	
		eState := E_CAC_DONE;

	(* complete *)
	E_CAC_DONE:

		(* no error found *)
		IF bError = FALSE THEN

			(* CAC data is valid *)
			bCACValid := TRUE;
			stCACData.CaseRejectCode 	:= 'OK';
			stCACData.CaseRejectID		:= 0;
		END_IF

		(* update outputs *)
		bBusy := FALSE;
		bDone := TRUE;
		strRejectCode := stCACData.CaseRejectCode;

		eState := E_CAC_IDLE;


(* unknown state *)
ELSE

	eState := E_CAC_IDLE;

	(* clear outputs *)
	bDone := FALSE;
	bBusy := FALSE;
	bError := FALSE;
	(*nErrorID := 0;*)
	bCACValid := FALSE;
END_CASE

END_FUNCTION_BLOCK

// ---- POUs/METS/Common LIB/08_SOFTWARE LIB/File FBs/FB_FILE_Move.TcPOU
(* move file(s) from SOURCE folder to TARGET folder, wildcard chars '*' and '?' can be used *)
FUNCTION_BLOCK FB_FILE_Move
VAR_INPUT
	bExecute			: BOOL;			(* set TRUE to copy multiple files *)
	strPathSource		: T_MaxString;	(* path of SOURCE folder *)
	strPathTarget		: T_MaxString;	(* path of TARGET folder *)
	strFileName			: T_MaxString;	(* file name to be moved, wildcard chars ('*', '?') can be used *)
	tTimeout			: TIME;			(* timeout for each file operation *)
END_VAR
VAR_OUTPUT
	bDone				: BOOL;			(* TRUE = file access complete *)
	bBusy				: BOOL;			(* TRUE = file access in progress *)
	bError				: BOOL;			(* TRUE = error occurred during process *)
	nErrorID			: UDINT;		(* error code *)
	strOutputFile		: T_MaxString;	(* name of file that failed *)
	strLastFileMoved		: T_MaxString;
END_VAR
VAR
	fbExecute			: R_TRIG;
	eState				: E_FILE_State;
	eErrorState			: E_FILE_State;
	fbFindFile			: FB_EnumFindFileEntry;
	eCommand			: E_EnumCmdType;
	strFoundFile		: T_MaxString;
	fbDeleteFile		: FB_FileDelete;
	fbMoveFile			: FB_FileRename;
END_VAR
(*
-------------------------------------------------------------------------------------------------
Date		Version	Author	Comments
-------------------------------------------------------------------------------------------------
30/01/2015	3.00.00	PB		Moved from Sewtec_CaseTrace.lib

-------------------------------------------------------------------------------------------------
27/09/2010	1.05.03	PB		If a file cannot be moved, FB will now continue to next file in list rather than just abort and report an error
							strOutputFile will contain the name of the last file that failed
23/03/2010	1.02.00	PB		Name changed from FB_FILE_MoveByByte to FB_FILE_Move
							Internal operation changed to delete target file (if exists) and move source file to target file using FB_FileRename
							Support for wildcard chars added to allow multiple files to be moved
02/03/2010	1.00.00	PB		Initial release

-------------------------------------------------------------------------------------------------
*)

(* compare files on rising edge of bExecute *)
fbExecute(CLK := bExecute);

CASE eState OF

	(* idle state *)
	E_FILE_IDLE:

		(* start new cycle *)
		IF fbExecute.Q = TRUE THEN

			(* reset outputs *)
			bDone := FALSE;
			bBusy := TRUE;
			bError := FALSE;
			nErrorID := 0;
			strOutputFile := '';
			strLastFileMoved :='';
			eErrorState := eState;

			(* start new file list *)
			eCommand := eEnumCmd_First;

			eState := E_FILE_FINDFILE;

		(* reset status outputs when no cycle is required and bExecute is reset *)
		ELSIF bExecute = FALSE THEN

			bDone := FALSE;
			bBusy := FALSE;
			bError := FALSE;
			nErrorID := 0;
			strOutputFile := '';
		END_IF


	(* find file *)
	E_FILE_FINDFILE:

		(* get file name *)
		fbFindFile(
			sNetId		:= '',
			sPathName	:= CONCAT(strPathSource, strFileName),
			eCmd		:= eCommand,
			bExecute	:= TRUE,
			tTimeout	:= T#1s,
		);

		(* find file complete *)
		IF fbFindFile.bBusy = FALSE THEN

			(* find file completed OK *)
			IF fbFindFile.bError = FALSE THEN

				(* file found *)
				IF fbFindFile.bEOE = FALSE THEN

					(* find next file in list *)
					eCommand := eEnumCmd_Next;

					(* ignore filenames '.' and '..' *)
					IF fbFindFile.stFindFile.sFileName <> '.' AND fbFindFile.stFindFile.sFileName <> '..' THEN

						strFoundFile := fbFindFile.stFindFile.sFileName;
						eState := E_FILE_DELETE;
					END_IF

				(* end of file list *)
				ELSE

					(* copy files complete *)
					eState := E_FILE_DONE;
				END_IF

			(* find file error *)
			ELSE

				(* no error has previously occurred *)
				IF bError = FALSE THEN

					(* log error code and failure state *)
					bError := TRUE;
					nErrorID := fbFindFile.nErrId;
					eErrorState := eState;
				END_IF

				(* abandon attempt to copy files *)
				eState := E_FILE_ABORT;
			END_IF

			(* close off fbFindFile *)
			fbFindFile(bExecute := FALSE);
		END_IF


	(* delete target file *)
	E_FILE_DELETE:

		(* delete file *)
		fbDeleteFile(
			sNetId		:= '',
			sPathName	:= CONCAT(strPathTarget, strFoundFile),
			ePath		:= PATH_GENERIC,
			bExecute	:= TRUE,
			tTimeout	:= tTimeout
		);

		(* file delete completed *)
		IF fbDeleteFile.bBusy = FALSE THEN

			(* file delete completed OK *)
			IF fbDeleteFile.bError = FALSE THEN

				eState := E_FILE_MOVE;

			(* file delete error *)
			ELSE

				(* file did not exist, OK to move file to TARGET folder *)
				IF fbDeleteFile.nErrId = 1804 THEN

					eState := E_FILE_MOVE;

				(* other file delete error occurred *)
				ELSE

					(* no error has previously occurred *)
					IF bError = FALSE THEN

						(* log error code and failure state *)
						strOutputFile := fbDeleteFile.sPathName;
						bError := TRUE;
						nErrorID := fbDeleteFile.nErrId;
						eErrorState := eState;
					END_IF

					(* move on to next file *)
					eState := E_FILE_FINDFILE;
				END_IF

			END_IF

			(* close off fbFileDelete *)
			fbDeleteFile(bExecute := FALSE);
		END_IF


	(* move source file to destination file *)
	E_FILE_MOVE:

		(* move file *)
		fbMoveFile(
			sNetId		:= '',
			sOldName	:= CONCAT(strPathSource, strFoundFile),
			sNewName	:= CONCAT(strPathTarget, strFoundFile),
			ePath		:= PATH_GENERIC,
			bExecute	:= TRUE,
			tTimeout	:= tTimeout,
		);
		
		(* file move completed *)
		IF fbMoveFile.bBusy = FALSE THEN

			(* file move completed OK *)
			IF fbMoveFile.bError = FALSE THEN

				strLastFileMoved :=strFoundFile;

			(* file move error *)
			ELSE

				(* no error has previously occurred *)
				IF bError = FALSE THEN

					(* log error code and failure state *)
					strOutputFile := fbMoveFile.sOldName;
					bError := TRUE;
					nErrorID := fbMoveFile.nErrId;
					eErrorState := eState;
				END_IF
			END_IF

			(* move on to next file *)
			eState := E_FILE_FINDFILE;

			(* close off fbMoveFile *)
			fbMoveFile(bExecute := FALSE);
		END_IF


	(* abort file entry list *)
	E_FILE_ABORT:

		(* abort file entry list *)
		fbFindFile(
			sNetId		:= '',
			sPathName	:= '',
			eCmd		:= eEnumCmd_Abort,
			bExecute	:= TRUE,
			tTimeout	:= T#1s,
		);

		(* abort file entry complete *)
		IF fbFindFile.bBusy = FALSE THEN

			(* abort file entry completed OK *)
			IF fbFindFile.bError = FALSE THEN

				eState := E_FILE_DONE;

			(* abort file entry error *)
			ELSE

				(* no error has previously occurred *)
				IF bError = FALSE THEN

					(* log error code and failure state *)
					bError := TRUE;
					nErrorID := fbFindFile.nErrId;
					eErrorState := eState;
				END_IF

				(* abandon attempt to copy files *)
				eState := E_FILE_DONE;
			END_IF

			(* close off fbFindFile *)
			fbFindFile(bExecute := FALSE);
		END_IF


	(* file access complete *)
	E_FILE_DONE:

		bDone := TRUE;
		bBusy := FALSE;

		(* return to IDLE state *)
		eState := E_FILE_IDLE;

END_CASE

END_FUNCTION_BLOCK

// ---- POUs/METS/Common LIB/02_OUTER LIB/Outer Functions/F_OUTER_BarcodeToHex.TcPOU
FUNCTION F_OUTER_BarcodeToHex : STRING(255)
VAR_INPUT
	strOuterBarcode		: T_OUTER_Barcode;
	stOuterCodeInfo						: ST_CodeInfo;
END_VAR
VAR

	strSerialCodeInHex	: STRING(255);
	nBarcodeLen	: INT;
	nCharIndex		: INT;
	nCharInDec		: BYTE;
	strCharInHex		: STRING(2);

	strChar			: STRING(1);
END_VAR

(* reset output *)
F_OUTER_BarcodeToHex := '';

 (*strSerialCodeInHex := F_OUTER_BarcodeToSerialCode(strOuterBarcode);*)
 strSerialCodeInHex := F_CODE_GetItem(strOuterBarcode, eCodeAIType.SerialCode, stOuterCodeInfo);

(* length of strPackCode *)
nBarcodeLen := LEN(strSerialCodeInHex);

(* strPackCode contains data *)
IF nBarcodeLen > 0 THEN

	(* check each char in the code *)
	FOR nCharIndex := 1 TO nBarcodeLen DO

		(* get char from string *)
		strChar := MID(strSerialCodeInHex, 1, nCharIndex);
		nCharInDec := F_ToASC(strChar);
		strCharInHex := DATA_TO_HEXSTR(ADR(nCharInDec), SIZEOF(nCharInDec), FALSE);
		F_OUTER_BarcodeToHex := CONCAT(F_OUTER_BarcodeToHex, strCharInHex);
	END_FOR
END_IF

END_FUNCTION

// ---- POUs/METS/Common LIB/08_SOFTWARE LIB/String FBs/F_CodeToHex.TcPOU
FUNCTION F_CodeToHex : T_MaxString
VAR_INPUT
	sCode		: T_MaxString;
END_VAR
VAR
	nCharIndex	: INT;
	sChar		: STRING(1);
	nCharInDec	: BYTE;
	sCharInHex	: STRING(2);

END_VAR

(* reset output *)
F_CodeToHex := '';

(* strPackCode contains data *)
IF LEN(sCode)  > 0  AND LEN(sCode) < 256 THEN

	(* check each char in the code *)
	FOR nCharIndex := 1 TO LEN(sCode)  DO

		(* get char from string *)
		sChar := MID(sCode, 1, nCharIndex);
		nCharInDec := F_ToASC(sChar);
		sCharInHex := DATA_TO_HEXSTR(ADR(nCharInDec), SIZEOF(nCharInDec), FALSE);
		F_CodeToHex := CONCAT(F_CodeToHex, sCharInHex);
	END_FOR

ELSIF LEN(sCode) >= 256 THEN
	F_CodeToHex :='Exceed_String_Length';
END_IF

END_FUNCTION

// ---- POUs/METS/Common LIB/08_SOFTWARE LIB/Counter FBs/FB_CTU32.TcPOU
(* 32-bit counter with count value as VAR_IN_OUT to allow count value to be set externally *)
FUNCTION_BLOCK FB_CTU32
VAR_INPUT
	bInput			: BOOL;		(* FALSE-TRUE increments counter value *)
	bReset			: BOOL;		(* set TRUE to reset counter value to 0 *)
	nThreshold		: UDINT;	(* threshold at which bOutput is set TRUE *)
END_VAR
VAR_IN_OUT
	nCounter		: UDINT;	(* counter value *)
END_VAR
VAR_OUTPUT
	bOutput			: BOOL;		(* nCounter >= nTheshold *)
END_VAR
VAR
	fbInputEdge		: R_TRIG;
END_VAR
(*
-------------------------------------------------------------------------------------------------
Date		Version	Author	Comments
-------------------------------------------------------------------------------------------------
30/01/2015	3.00.00	PB		No change

-------------------------------------------------------------------------------------------------
05/02/10	1.00.00	PB		Initial release

-------------------------------------------------------------------------------------------------
*)

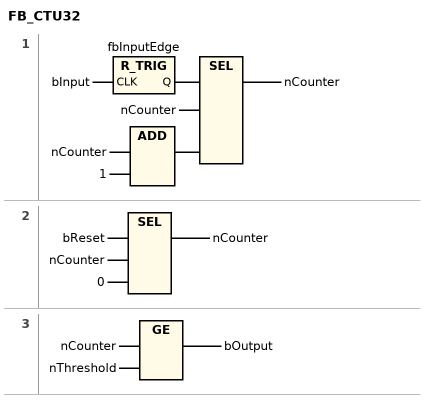
// NETWORK 1
fbInputEdge(CLK := bInput); // R_TRIG
nCounter := SEL(fbInputEdge.Q, nCounter, nCounter + 1);

// NETWORK 2
nCounter := SEL(bReset, nCounter, 0);

// NETWORK 3
bOutput := nCounter >= nThreshold;

END_FUNCTION_BLOCK

// ---- POUs/METS/Common LIB/08_SOFTWARE LIB/Debug/FB_DEBUG_CounterArray.TcPOU
FUNCTION_BLOCK FB_DEBUG_CounterArray
(* Array of CU in one function block for tidyier debugging. *)
VAR_INPUT
	CU1					: BOOL;
	CU2					: BOOL;
	CU3					: BOOL;
	CU4					: BOOL;
	CU5					: BOOL;
	CU6					: BOOL;
	CU7					: BOOL;	(*  *)
	CU8					: BOOL;
	CU9					: BOOL;
	CU10				: BOOL;
	PV					: WORD;
	bReset				: BOOL;
END_VAR
VAR_OUTPUT
	CV1					: UINT;
	CV2					: UINT;
	CV3					: UINT;
	CV4					: UINT;
	CV5					: UINT;
	CV6					: UINT;
	CV7					: UINT;
	CV8					: UINT;
	CV9					: UINT;
	CV10				: UINT;
END_VAR
VAR
	aCTU				: ARRAY [1..10] OF CTU;
END_VAR

aCTU[1](CU := CU1, RESET := bReset, PV := PV, CV => CV1);
aCTU[2](CU := CU2, RESET := bReset, PV := PV, CV => CV2);
aCTU[3](CU := CU3, RESET := bReset, PV := PV, CV => CV3);
aCTU[4](CU := CU4, RESET := bReset, PV := PV, CV => CV4);
aCTU[5](CU := CU5, RESET := bReset, PV := PV, CV => CV5);
aCTU[6](CU := CU6, RESET := bReset, PV := PV, CV => CV6);
aCTU[7](CU := CU7, RESET := bReset, PV := PV, CV => CV7);
aCTU[8](CU := CU8, RESET := bReset, PV := PV, CV => CV8);
aCTU[9](CU := CU9, RESET := bReset, PV := PV, CV => CV9);
aCTU[10](CU := CU10, RESET := bReset, PV := PV, CV => CV10);

END_FUNCTION_BLOCK

// ---- POUs/METS/Common LIB/04_CASE LIB/Case Functons/F_CASE_ClearCurrentPackerData.TcPOU
(* clear all data from Packer Data  *)
FUNCTION F_CASE_ClearCurrentPackerData : BOOL
VAR_INPUT
	bEnable				: BOOL;			(* set TRUE to reset all values in Packer Data *)
END_VAR

VAR_IN_OUT
	stCurrentPackerData					: ST_CASE_OperationData;
END_VAR

(* clear Packer Data  enabled *)
IF bEnable = TRUE THEN

	(* reset Packer Data  *)
	MEMSET(ADR(stCurrentPackerData), 16#00, SIZEOF(stCurrentPackerData));

	(* set output to TRUE when reset is active *)
	F_CASE_ClearCurrentPackerData := TRUE;

(* clear Packer Data  disabled *)
ELSE

	(* reset output *)
	F_CASE_ClearCurrentPackerData := FALSE;
END_IF

END_FUNCTION

// ---- POUs/_Exclude/FB_SYSTEM_CheckOS.TcPOU
(* reads a registry key to determine if OS is WinCE or full Windows *)
FUNCTION_BLOCK FB_SYSTEM_CheckOS
VAR_INPUT
	bExecute		: BOOL;		(* check OS type *)
END_VAR
VAR_OUTPUT
	bDone			: BOOL;		(* TRUE = OS check complete *)
	bBusy 			: BOOL;		(* TRUE = OS check active *)
	bError			: BOOL;		(* TRUE = OS check error *)
	nErrorID		: UDINT;	(* error code *)
	eOSType			: E_SYSTEM_OSType;	(* OS type *)
END_VAR
VAR
	fbExecute		: R_TRIG;
	nState			: INT;
	strData			: STRING(255);
	fbReadRegKey	: FB_RegQueryValue;
END_VAR
(*
-------------------------------------------------------------------------------------------------
Date		Version	Author	Comments
-------------------------------------------------------------------------------------------------
30/01/2015	3.00.00	PB		Initial release

-------------------------------------------------------------------------------------------------
*)

(* monitor bExecute *)
fbExecute(CLK := bExecute);

CASE nState OF

	(* idle *)
	0:

		(* rising edge on bExecute *)
		IF fbExecute.Q = TRUE THEN

			(* reset status outputs *)
			bDone := FALSE;
			bBusy := TRUE;
			bError := FALSE;
			nErrorID := 0;

			(* reset vars *)
			eOSType := E_OS_UNKNOWN;
			MEMSET(ADR(strData), 16#00, SIZEOF(strData));

			nState := 1;

		(* bExecute has been reset *)
		ELSIF bExecute = FALSE THEN

			(* reset status outputs *)
			bDone := FALSE;
			bBusy := FALSE;
			bError := FALSE;
			nErrorID := 0;
		END_IF


	(* read registry *)
	1:

		(* read registry key *)
		fbReadRegKey(
			sNetId		:= '',
			sSubKey		:= 'SOFTWARE\Beckhoff\TwinCAT',
			sValName	:= 'InstallationPath',
			cbData		:= SIZEOF(strData),
			pData		:= ADR(strData),
			bExecute	:= TRUE,
			tTimeOut	:= T#1s
		);

		(* read registry key complete *)
		IF fbReadRegKey.bBusy = FALSE THEN

			(* read registry key completed OK *)
			IF fbReadRegKey.bError = FALSE THEN

				(* value on WinCE will be '\Hard Disk\TwinCAT' *)
				IF strData = '\Hard Disk\TwinCAT' THEN

					(* OS is WinCE *)
					eOSType := E_OS_WINCE;

				(* other value *)
				ELSE

					(* OS is full Windows *)
					eOSType := E_OS_WINDOWS;
				END_IF

			(* read registry key error *)
			ELSE

				(* update outputs *)
				bError := TRUE;
				nErrorID := fbReadRegKey.nErrId;
			END_IF

			nState := 20;

			(* close off fbReadRegKey *)
			fbReadRegKey(bExecute := FALSE);
		END_IF


	(* done *)
	20:

		(* update status outputs *)
		bDone := TRUE;
		bBusy := FALSE;

		nState := 0;


(* unknown state *)
ELSE

	nState := 0;
END_CASE

END_FUNCTION_BLOCK

// ---- POUs/_Exclude/FB_SYSTEM_CreateFolders.TcPOU
FUNCTION_BLOCK FB_SYSTEM_CreateFolders
VAR_INPUT
	bExecute				: BOOL;		(* set TRUE to generate system folders *)
	sBasePath			: T_FolderName;	(* CaseTrace base folder path *)
	aBaseFolder			: ARRAY[1..cSYSTEM_FOLDER_LIMIT] OF T_FolderName;
END_VAR
VAR_OUTPUT
	bDone				: BOOL;		(* TRUE = system folders complete *)
	bBusy				: BOOL;		(* TRUE = system folders in progress *)
	bError				: BOOL;		(* TRUE = system folders error *)
	nErrorID				: UDINT;	(* error code *)
	bSystemFolderOK		: BOOL;		(* TRUE = system folders OK *)
	sStatus					: STRING(25);	(* system folder status *)
	sLocalArchiveDBPath		: T_FolderPath;	(*local ArchiveDB path*)
	sLocalBridgePath 			: T_FolderPath;	(* local Bridge path *)
	sLocalPCMPath 			: T_FolderPath;	(* local PCM path *)
	sLocalPCMIncomingPath 	: T_FolderPath;	(* local PCM/Incoming path *)
	sLocalOCVPath 			: T_FolderPath;	(* local OCV path *)
	sLocalOACPath 			: T_FolderPath;	(* local OAC path *)
	sLocalCACPath 			: T_FolderPath;	(* local CAC path *)
	sLocalPACPath 			: T_FolderPath;	(* local PAC path *)
	sLocalOHMPath 			: T_FolderPath;	(* local OHM path *)
	sLocalCHMPath 			: T_FolderPath;	(* local CHM path *)
	sLocalPHMPath			: T_FolderPath;	(* local PHM path *)
	sLocalKPIPath 			: T_FolderPath;	(* local KPI path *)
	sLocalHMIPath 			: T_FolderPath;	(* local HMI path *)
	sLocalSettingsPath		 	: T_FolderPath;	(* local Setting*)
	sLocalBackupsPath			: T_FolderPath; (*local Setting/Backup path*)
	sLocalTemplatesPath		: T_FolderPath;	(* local Templates path *)
	sLocalOrcaPath			: T_FolderPath;	(* local Orca path *)
	sLocalSystemLogPath			: T_FolderPath;	(* local Log path *)
	sLocaCameraPath			: T_FolderPath;	(* local Camera path *)

END_VAR
VAR
	fbExecute				: R_TRIG;
	eState				: E_SYSTEM_MaintainFolders;
	eErrorState			: E_SYSTEM_MaintainFolders;
	nMaxIndex			: INT;
	nIndex				: INT;
	eCmdType		: E_EnumCmdType;
	fbFindFolder		: FB_EnumFindFileEntry;
	fbCreateFolder			: FB_CreateDir;

END_VAR

(* rising edge of bExecute *)
fbExecute(CLK := bExecute);

CASE eState OF

	(* idle *)
	E_FOLDER_IDLE:

		(* rising edge of bExecute *)
		IF fbExecute.Q = TRUE THEN

			(* update outputs *)
			bDone := FALSE;
			bBusy := TRUE;
			bError := FALSE;
			nErrorID := 0;

			(* max number of BASE folders and start with 1st folder *)
			nMaxIndex := UDINT_TO_INT(SIZEOF(aBaseFolder) / SIZEOF(aBaseFolder[1]));
			nIndex := 1;
			eCmdType := eEnumCmd_First;

			//eState := E_FOLDER_CREATEBASEPATH;
			eState := E_FOLDER_ININT_CHECK;

		(* bExecute has been reset *)
		ELSIF bExecute = FALSE THEN

			(* reset outputs *)
			bDone := FALSE;
			bBusy := FALSE;
			bError := FALSE;
			nErrorID := 0;
		END_IF

	E_FOLDER_ININT_CHECK:
					eCmdType := eEnumCmd_First;
					eState := E_FOLDER_CHECK;
	
	E_FOLDER_CHECK:

		(* find folder *)
		fbFindFolder(
			sNetId		:= '',
			sPathName	:= CONCAT(sBasePath, aBaseFolder[nIndex]),
			eCmd		:= eCmdType,
			bExecute	:= TRUE,
			tTimeout	:= T#1s
		);

		(* find folder complete *)
		IF fbFindFolder.bBusy = FALSE THEN

			(* find folder completed OK *)
			IF fbFindFolder.bError = FALSE THEN

				(* folder found *)
				IF fbFindFolder.stFindFile.fileAttributes.bDirectory = TRUE THEN

				
						(* all BASE folders completed *)
				IF nIndex = nMaxIndex THEN

					eState := E_FOLDER_DONE;

				(* more BASE folders *)
				ELSE
					nIndex := nIndex + 1;
					eCmdType := eEnumCmd_Abort;
					eState := E_FOLDER_ININT_CHECK;
				END_IF

				(* end of list *)
				ELSIF fbFindFolder.bEOE = TRUE THEN

						eState := E_FOLDER_CREATEBASEPATH;
				END_IF

			(* find folder completed OK *)
			ELSE

				(* update outputs *)
				bError := TRUE;
				nErrorID := fbFindFolder.nErrID;
				eErrorState := eState;

				eState := E_FOLDER_DONE;
			END_IF

			(* close off fbFindFolder *)
			fbFindFolder(bExecute := FALSE);
		END_IF
		
	(* create BASE folders *)
	E_FOLDER_CREATEBASEPATH:

		(* create folder *)
		fbCreateFolder(
			sNetId		:= '',
			sPathName	:= CONCAT(sBasePath, aBaseFolder[nIndex]),
			ePath		:= PATH_GENERIC,
			bExecute	:= TRUE,
			tTimeout	:= T#1s
		);

		(* create folder complete *)
		IF fbCreateFolder.bBusy = FALSE THEN

			(* create folder completed OK or folder already exists *)
			IF fbCreateFolder.bError = FALSE OR (fbCreateFolder.bError = TRUE AND fbCreateFolder.nErrId = cFAILED_OBJECT_ALREADY_EXIST) THEN

				(* all BASE folders completed *)
				IF nIndex = nMaxIndex THEN

					eState := E_FOLDER_DONE;

				(* more BASE folders *)
				ELSE

					(* next BASE folder *)
					nIndex := nIndex + 1;
					eState := E_FOLDER_ININT_CHECK;
				END_IF

			(* create folder error *)
			ELSE

				(* no error active *)
				IF bError = FALSE THEN

					(* update outputs *)
					bError := TRUE;
					nErrorID := fbCreateFolder.nErrId;
					eErrorState := eState;
					sStatus := CONCAT(sBasePath, aBaseFolder[nIndex]);
				END_IF

				eState := E_FOLDER_DONE;
			END_IF

			(* close off fbCreateFolder *)
			fbCreateFolder(bExecute := FALSE);
		END_IF


	(* done *)
	E_FOLDER_DONE:

		(* no error occurred *)
		IF bError = FALSE THEN

			(* update status *)
			bSystemFolderOK 		:= TRUE;
			sStatus 				:= 'Folders OK';

			(* populate local folder paths *)
			sLocalBridgePath		:= CONCAT(sBasePath, aBaseFolder[1]);
			sLocalPCMPath 		:= CONCAT(sBasePath, aBaseFolder[28]);
			sLocalPCMIncomingPath		:= CONCAT(sBasePath, aBaseFolder[31]);
			sLocalOCVPath 		:= CONCAT(sBasePath, aBaseFolder[21]);
			sLocalOACPath 		:= CONCAT(sBasePath, aBaseFolder[19]);
			sLocalCACPath 		:= CONCAT(sBasePath, aBaseFolder[4]);
			sLocalPACPath 		:= CONCAT(sBasePath, aBaseFolder[32]);
			sLocalOHMPath 		:= CONCAT(sBasePath, aBaseFolder[23]);
			sLocalCHMPath		:= CONCAT(sBasePath, aBaseFolder[9]);
			sLocalPHMPath		:= CONCAT(sBasePath, aBaseFolder[33]);
			sLocalKPIPath 		:= CONCAT(sBasePath, aBaseFolder[15]);
			sLocalHMIPath	 	:= CONCAT(sBasePath, aBaseFolder[14]);
			sLocalSettingsPath 		:= CONCAT(sBasePath, aBaseFolder[37]);
			sLocalBackupsPath 	:= CONCAT(sBasePath, aBaseFolder[38]);
			sLocalTemplatesPath	:= CONCAT(sBasePath, aBaseFolder[39]);
			sLocalOrcaPath		:= CONCAT(sBasePath, aBaseFolder[40]);
			sLocalSystemLogPath		:= CONCAT(sBasePath, aBaseFolder[41]);
			sLocaCameraPath		:= CONCAT(sBasePath, aBaseFolder[42]);
			sLocalArchiveDBPath		:= CONCAT(sBasePath, aBaseFolder[43]);

		(* else *)
		ELSE

			(* clear local paths *)
			sLocalBridgePath := '';
			sLocalPCMPath := '';
			sLocalPCMIncomingPath	:= '';
			sLocalOCVPath := '';
			sLocalOACPath := '';
			sLocalCACPath := '';
			sLocalPACPath := '';
			sLocalOHMPath := '';
			sLocalCHMPath := '';
			sLocalPHMPath := '';
			sLocalKPIPath := '';
			sLocalHMIPath := '';
			sLocalSettingsPath 	:= '';
			sLocalBackupsPath :='';
			sLocalTemplatesPath :='';
			sLocalOrcaPath :='';
			sLocalSystemLogPath	:='';
			sLocaCameraPath		:='';
			sLocalArchiveDBPath	:='';
		END_IF

		(* update outputs *)
		bDone := TRUE;
		bBusy := FALSE;

		eState := E_FOLDER_IDLE;


(* unknown state *)
ELSE

	eState := E_FOLDER_IDLE;

	(* reset outputs *)
	bDone := FALSE;
	bBusy := FALSE;
	bError := FALSE;
	nErrorID := 0;
	bSystemFolderOK := FALSE;
	sStatus := '';
	sLocalBridgePath := '';
	sLocalPCMPath := '';
	sLocalPCMIncomingPath	:= '';
	sLocalOCVPath := '';
	sLocalOACPath := '';
	sLocalCACPath := '';
	sLocalPACPath := '';
	sLocalOHMPath := '';
	sLocalCHMPath := '';
	sLocalPHMPath := '';
	sLocalKPIPath := '';
	sLocalHMIPath := '';
	sLocalSettingsPath 	:= '';
	sLocalBackupsPath :='';
	sLocalTemplatesPath :='';
	sLocalOrcaPath :='';
	sLocalSystemLogPath	:='';
	sLocaCameraPath		:='';
	sLocalArchiveDBPath	:='';
END_CASE

END_FUNCTION_BLOCK

// ---- POUs/METS/Common LIB/01_PACK LIB/OCV FBs/FB_OCV_FindDB.TcPOU
(* converts strOuterBarcode to OCV filename and loads data *)
FUNCTION_BLOCK FB_OCV_FindDB
VAR_INPUT
	bExecute				: BOOL;		(* set TRUE to load OCV file *)
	sPackBarcode			: T_PACK_Barcode;	(* Outer barcode *)
	nAcceptanceLevel			: INT;
	bUseInterimCodeForValidation	: BOOL;
END_VAR
VAR_IN_OUT
	stOCVDataDB							: ST_DB_OCVDataCtrl;
	stCodeInfo_Pack				: ST_CodeInfo;
	stCodeInfo_Intermediate		: ST_CodeInfo;
END_VAR
VAR_OUTPUT
	bDone				: BOOL;		(* TRUE = find file complete *)
	bBusy				: BOOL;		(* TRUE = find file in progress *)
	bError				: BOOL;		(* TRUE = error occurred *)
	nErrorID				: UDINT;		(* error code *)
	bOCVDataFound		: BOOL;		(* TRUE = OCV file found *)
	bOCVDataValid		: BOOL;		(* TRUE - OCV file valide*)
	aOCVRecordDBName			 : ARRAY[1..2] OF T_MaxString;
END_VAR
VAR
	fbExecute				: R_TRIG;
	eState				: E_OCV_State;
	eErrorState				: E_OCV_State;
	eCodeAIType				: E_CodeAIType;


	tonTimeOut				: TON;
	rtTimeOutExec				: R_TRIG;

	stOCVData			: ST_OUTER_Status;
END_VAR

(***************************************TimeOut *******************************************)
(* monitor Busy timeout *)
tonTimeOut( IN:=eState=E_OCV_DBREQUEST, PT:=cTHREE_SECONDS, Q=>);
(*	cTHREE_SECONDS						: TIME := T#3s;
	cFIVE_SECONDS						: TIME := t#5s;
	cTEN_SECONDS						: TIME := t#10s;*)

rtTimeOutExec(CLK:= tonTimeOut.Q);

IF rtTimeOutExec.Q THEN

	bError := TRUE;
	nErrorID := 100;
	eErrorState := eState;

	MEMSET(ADR(stOCVDataDB), 16#00, SIZEOF(stOCVDataDB));

	eState := E_OCV_DONE;
END_IF

(***************************************Execution*******************************************)

fbExecute(CLK := bExecute);

CASE eState OF

	(* idle *)
	E_OCV_IDLE:

		(* rising edge of bExecute *)
		IF fbExecute.Q = TRUE THEN

			(* initialise outputs *)
			bDone := FALSE;
			bBusy := TRUE;
			bError := FALSE;
			nErrorID := 0;

			MEMSET(ADR(aOCVRecordDBName), 16#00, SIZEOF(aOCVRecordDBName));
			(* convert strOuterBarcode to OAC filename *)
			bOCVDataFound := FALSE;
			bOCVDataValid := FALSE;
			MEMSET(ADR(stOCVData), 16#00, SIZEOF(stOCVData));

			eState := E_OCV_DBREQUEST;

		(* bExecute has been reset *)
		ELSIF bExecute = FALSE THEN

			(* reset outputs *)
			bDone := FALSE;
			bBusy := FALSE;
			bError := FALSE;
			(*nErrorID := 0;*)

			(*bOCVFileFound := FALSE;*)
			(*bOCVFileValide := FALSE;*)
		END_IF

	E_OCV_DBREQUEST:

		stOCVDataDB.bReadDataReq		:=TRUE;

		IF F_InvalidateASCIIChar(F_CODE_GetItem(sPackBarcode , eCodeAIType.SerialCode,
													SEL(bUseInterimCodeForValidation  , stCodeInfo_Pack, stCodeInfo_Intermediate))) =	0 	THEN

			stOCVDataDB.sFileCodeName1	:= F_CodeToHex(F_CODE_GetItem(sPackBarcode , eCodeAIType.SerialCode,
													SEL(bUseInterimCodeForValidation  , stCodeInfo_Pack, stCodeInfo_Intermediate)));
		END_IF

(*place for HectorDB block*)

		IF stOCVDataDB.bDone THEN
			IF NOT stOCVDataDB.bError THEN		(* f.ex not found, or DB transaction faild??*)

				stOCVData := stOCVDataDB.stOCVStatusDB;
				aOCVRecordDBName[1] := stOCVDataDB.stOCVStatusDB.stOACData.AggregationCodes[1];
				aOCVRecordDBName[2] := stOCVDataDB.stOCVStatusDB.stOACData.AggregationCodes[2];
				(* OCV record exists *)
				bOCVDataFound := TRUE;

				IF stOCVData.stOACData.NumberOfLinkedPacks >= nAcceptanceLevel THEN
					bOCVDataValid := TRUE;
				END_IF
			ELSE
				bError := TRUE;
				nErrorID := stOCVDataDB.nErrorID;

				eErrorState := eState;
			END_IF

			MEMSET(ADR(stOCVDataDB), 16#00, SIZEOF(stOCVDataDB));

			eState := E_OCV_DONE;
		END_IF


	(* complete *)
	E_OCV_DONE:

		(* update outputs *)
		bDone := TRUE;
		bBusy := FALSE;

		eState := E_OCV_IDLE;

(* unknown state *)
ELSE

	eState := E_OCV_IDLE;

	(* clear outputs *)
	bDone := FALSE;
	bBusy := FALSE;
	bError := FALSE;
	(*nErrorID := 0;*)

END_CASE

END_FUNCTION_BLOCK

// ---- POUs/METS/Common LIB/08_SOFTWARE LIB/String FBs/F_InvalidateASCIIChar.TcPOU
FUNCTION F_InvalidateASCIIChar : INT
VAR_INPUT
	sCode		: STRING(255);
END_VAR
VAR
	nCodeLen	: INT;
	nCharIndex		: INT;
	sChar			: STRING(1);
END_VAR

(* reset output *)
F_InvalidateASCIIChar := 0;

(* strPackCode contains data *)
IF LEN(sCode) = 0 THEN

	F_InvalidateASCIIChar := -1;

ELSIF LEN(sCode) > 0 THEN

	(* check each char in the code *)
	FOR nCharIndex := 1 TO LEN(sCode) DO

		(* get char from string *)
		sChar := MID(sCode, 1, nCharIndex);

		(* check if every char valid for proccessig*)
		IF (F_ToASC(sChar) < 16#21 OR  F_ToASC(sChar) >  16#7A) AND   F_ToASC(sChar) <> 16#7C THEN	(*  16#7C -> '|'*)

			(* update valid char counter *)
			F_InvalidateASCIIChar := F_InvalidateASCIIChar + 1;
		END_IF
	END_FOR
END_IF

END_FUNCTION

// ---- POUs/METS/Common LIB/01_PACK LIB/Pack FBs/FB_PACK_DuplicatesPackCodesDB.TcPOU
FUNCTION_BLOCK FB_PACK_DuplicatesPackCodesDB
VAR_INPUT
	stDuplicatedItem						: ST_RejectItems;
	nMaxOuterIndex					: INT;
	nSourceIndex						: INT;
	bExtendedDupCheck					: BOOL;
END_VAR
VAR_OUTPUT
	bDuplicateFound 				: BOOL;
END_VAR
VAR_IN_OUT
	stOuterStatus				: ST_OUTER_Status;	(* Outer status *)
	stLastOuterStatus			: ST_OUTER_Status;	(* Outer status *)
END_VAR
VAR
	nCheckIndex : T_PositiveINT;
	nPackIndex : T_PositiveINT;

	nGoodPackReads	: T_PositiveINT;
END_VAR

(* for dupicats for packs in next  Outer in queue*)		(*nSourceIndex cannot be equal cMAX_OUTER_STATUS_QUEUE because input data will be out of index*)
IF	bExtendedDupCheck AND stLastOuterStatus.nStatus.6 AND nSourceIndex < cMAX_OUTER_STATUS_QUEUE THEN
	(* for all other Packs in Outer *)
	FOR  nPackIndex :=1 TO cMAX_PACKS_PER_OUTER DO

